LIN {X 72.334,Y 67.048,Z 77.329,A 180.000,B 0.000,C 180.000} C_DIS
LIN {X 72.380,Y 66.990,Z 77.327,A 180.000,B 0.000,C 180.000} C_DIS
LIN {X 72.424,Y 66.930,Z 77.324,A 180.000,B 0.000,C 180.000} C_DIS
LIN {X 72.502,Y 66.814,Z 77.319,A 180.000,B 0.000,C 180.000} C_DIS
LIN {X 72.574,Y 66.694,Z 77.315,A 180.000,B 0.000,C 180.000} C_DIS
LIN {X 72.610,Y 66.630,Z 77.312,A 180.000,B 0.000,C 180.000} C_DIS
LIN {X 72.644,Y 66.564,Z 77.309,A 180.000,B 0.000,C 180.000} C_DIS
LIN {X 72.676,Y 66.497,Z 77.307,A 180.000,B 0.000,C 180.000} C_DIS
LIN {X 72.706,Y 66.429,Z 77.304,A 180.000,B 0.000,C 180.000} C_DIS
LIN {X 72.757,Y 66.302,Z 77.299,A 180.000,B 0.000,C 180.000} C_DIS
LIN {X 72.800,Y 66.173,Z 77.295,A 180.000,B 0.000,C 180.000} C_DIS
LIN {X 72.838,Y 66.038,Z 77.290,A 180.000,B 0.000,C 180.000} C_DIS
LIN {X 72.869,Y 65.902,Z 77.285,A 180.000,B 0.000,C 180.000} C_DIS
LIN {X 72.882,Y 65.831,Z 77.282,A 180.000,B 0.000,C 180.000} C_DIS
LIN {X 72.893,Y 65.760,Z 77.280,A 180.000,B 0.000,C 180.000} C_DIS
LIN {X 72.901,Y 65.688,Z 77.277,A 180.000,B 0.000,C 180.000} C_DIS
LIN {X 72.908,Y 65.617,Z 77.275,A 180.000,B 0.000,C 180.000} C_DIS
LIN {X 72.916,Y 65.480,Z 77.270,A 180.000,B 0.000,C 180.000} C_DIS
LIN {X 72.916,Y 65.344,Z 77.265,A 180.000,B 0.000,C 180.000} C_DIS
LIN {X 72.909,Y 65.208,Z 77.261,A 180.000,B 0.000,C 180.000} C_DIS
LIN {X 72.895,Y 65.072,Z 77.256,A 180.000,B 0.000,C 180.000} C_DIS
LIN {X 72.873,Y 64.933,Z 77.251,A 180.000,B 0.000,C 180.000} C_DIS
LIN {X 72.842,Y 64.795,Z 77.246,A 180.000,B 0.000,C 180.000} C_DIS
LIN {X 72.823,Y 64.722,Z 77.243,A 180.000,B 0.000,C 180.000} C_DIS
LIN {X 72.802,Y 64.649,Z 77.241,A 180.000,B 0.000,C 180.000} C_DIS
LIN {X 72.759,Y 64.503,Z 77.235,A 180.000,B 0.000,C 180.000} C_DIS
LIN {X 72.737,Y 64.427,Z 77.233,A 180.000,B 0.000,C 180.000} C_DIS
LIN {X 72.715,Y 64.352,Z 77.230,A 180.000,B 0.000,C 180.000} C_DIS
LIN {X 72.693,Y 64.276,Z 77.227,A 180.000,B 0.000,C 180.000} C_DIS
LIN {X 72.670,Y 64.201,Z 77.224,A 180.000,B 0.000,C 180.000} C_DIS
LIN {X 72.648,Y 64.125,Z 77.222,A 180.000,B 0.000,C 180.000} C_DIS
LIN {X 72.626,Y 64.049,Z 77.219,A 180.000,B 0.000,C 180.000} C_DIS
LIN {X 72.604,Y 63.974,Z 77.216,A 180.000,B 0.000,C 180.000} C_DIS
LIN {X 72.582,Y 63.898,Z 77.213,A 180.000,B 0.000,C 180.000} C_DIS
LIN {X 72.560,Y 63.822,Z 77.211,A 180.000,B 0.000,C 180.000} C_DIS
LIN {X 72.537,Y 63.747,Z 77.208,A 180.000,B 0.000,C 180.000} C_DIS
LIN {X 72.515,Y 63.671,Z 77.205,A 180.000,B 0.000,C 180.000} C_DIS
LIN {X 72.493,Y 63.596,Z 77.202,A 180.000,B 0.000,C 180.000} C_DIS
LIN {X 72.471,Y 63.520,Z 77.200,A 180.000,B 0.000,C 180.000} C_DIS
LIN {X 72.449,Y 63.444,Z 77.197,A 180.000,B 0.000,C 180.000} C_DIS
LIN {X 72.427,Y 63.369,Z 77.194,A 180.000,B 0.000,C 180.000} C_DIS
LIN {X 72.404,Y 63.293,Z 77.191,A 180.000,B 0.000,C 180.000} C_DIS
LIN {X 72.382,Y 63.217,Z 77.189,A 180.000,B 0.000,C 180.000} C_DIS
LIN {X 72.360,Y 63.142,Z 77.186,A 180.000,B 0.000,C 180.000} C_DIS
LIN {X 72.338,Y 63.066,Z 77.183,A 180.000,B 0.000,C 180.000} C_DIS
LIN {X 72.316,Y 62.991,Z 77.180,A 180.000,B 0.000,C 180.000} C_DIS
LIN {X 72.293,Y 62.915,Z 77.178,A 180.000,B 0.000,C 180.000} C_DIS
LIN {X 72.271,Y 62.839,Z 77.175,A 180.000,B 0.000,C 180.000} C_DIS
LIN {X 72.249,Y 62.764,Z 77.172,A 180.000,B 0.000,C 180.000} C_DIS
LIN {X 72.227,Y 62.688,Z 77.170,A 180.000,B 0.000,C 180.000} C_DIS
LIN {X 72.204,Y 62.613,Z 77.167,A 180.000,B 0.000,C 180.000} C_DIS
LIN {X 72.182,Y 62.537,Z 77.165,A 180.000,B 0.000,C 180.000} C_DIS
LIN {X 72.160,Y 62.461,Z 77.162,A 180.000,B 0.000,C 180.000} C_DIS
LIN {X 72.137,Y 62.386,Z 77.159,A 180.000,B 0.000,C 180.000} C_DIS
LIN {X 72.115,Y 62.310,Z 77.157,A 180.000,B 0.000,C 180.000} C_DIS
LIN {X 72.093,Y 62.235,Z 77.154,A 180.000,B 0.000,C 180.000} C_DIS
LIN {X 72.070,Y 62.159,Z 77.152,A 180.000,B 0.000,C 180.000} C_DIS
LIN {X 72.048,Y 62.084,Z 77.149,A 180.000,B 0.000,C 180.000} C_DIS
LIN {X 72.003,Y 61.932,Z 77.144,A 180.000,B 0.000,C 180.000} C_DIS
LIN {X 71.958,Y 61.781,Z 77.139,A 180.000,B 0.000,C 180.000} C_DIS
LIN {X 71.913,Y 61.630,Z 77.134,A 180.000,B 0.000,C 180.000} C_DIS
LIN {X 71.868,Y 61.479,Z 77.130,A 180.000,B 0.000,C 180.000} C_DIS
LIN {X 71.823,Y 61.328,Z 77.125,A 180.000,B 0.000,C 180.000} C_DIS
LIN {X 71.777,Y 61.177,Z 77.120,A 180.000,B 0.000,C 180.000} C_DIS
LIN {X 71.732,Y 61.027,Z 77.116,A 180.000,B 0.000,C 180.000} C_DIS
LIN {X 71.687,Y 60.876,Z 77.111,A 180.000,B 0.000,C 180.000} C_DIS
LIN {X 71.641,Y 60.725,Z 77.107,A 180.000,B 0.000,C 180.000} C_DIS
LIN {X 71.596,Y 60.574,Z 77.102,A 180.000,B 0.000,C 180.000} C_DIS
LIN {X 71.550,Y 60.423,Z 77.098,A 180.000,B 0.000,C 180.000} C_DIS
LIN {X 71.504,Y 60.272,Z 77.094,A 180.000,B 0.000,C 180.000} C_DIS
LIN {X 71.458,Y 60.122,Z 77.090,A 180.000,B 0.000,C 180.000} C_DIS
LIN {X 71.412,Y 59.971,Z 77.086,A 180.000,B 0.000,C 180.000} C_DIS
LIN {X 71.366,Y 59.820,Z 77.082,A 180.000,B 0.000,C 180.000} C_DIS
LIN {X 71.320,Y 59.669,Z 77.078,A 180.000,B 0.000,C 180.000} C_DIS
LIN {X 71.274,Y 59.519,Z 77.074,A 180.000,B 0.000,C 180.000} C_DIS
LIN {X 71.228,Y 59.368,Z 77.070,A 180.000,B 0.000,C 180.000} C_DIS
LIN {X 71.182,Y 59.218,Z 77.066,A 180.000,B 0.000,C 180.000} C_DIS
LIN {X 71.135,Y 59.067,Z 77.063,A 180.000,B 0.000,C 180.000} C_DIS
LIN {X 71.089,Y 58.917,Z 77.059,A 180.000,B 0.000,C 180.000} C_DIS
LIN {X 71.042,Y 58.766,Z 77.056,A 180.000,B 0.000,C 180.000} C_DIS
LIN {X 70.995,Y 58.616,Z 77.053,A 180.000,B 0.000,C 180.000} C_DIS
LIN {X 70.948,Y 58.465,Z 77.049,A 180.000,B 0.000,C 180.000} C_DIS
LIN {X 70.901,Y 58.315,Z 77.046,A 180.000,B 0.000,C 180.000} C_DIS
LIN {X 70.854,Y 58.164,Z 77.043,A 180.000,B 0.000,C 180.000} C_DIS
LIN {X 70.807,Y 58.014,Z 77.040,A 180.000,B 0.000,C 180.000} C_DIS
LIN {X 70.760,Y 57.864,Z 77.037,A 180.000,B 0.000,C 180.000} C_DIS
LIN {X 70.713,Y 57.714,Z 77.035,A 180.000,B 0.000,C 180.000} C_DIS
LIN {X 70.665,Y 57.563,Z 77.032,A 180.000,B 0.000,C 180.000} C_DIS
LIN {X 70.618,Y 57.413,Z 77.029,A 180.000,B 0.000,C 180.000} C_DIS
LIN {X 70.570,Y 57.263,Z 77.027,A 180.000,B 0.000,C 180.000} C_DIS
LIN {X 70.474,Y 56.963,Z 77.022,A 180.000,B 0.000,C 180.000} C_DIS
LIN {X 70.378,Y 56.663,Z 77.018,A 180.000,B 0.000,C 180.000} C_DIS
LIN {X 70.282,Y 56.363,Z 77.014,A 180.000,B 0.000,C 180.000} C_DIS
LIN {X 70.185,Y 56.063,Z 77.011,A 180.000,B 0.000,C 180.000} C_DIS
LIN {X 70.087,Y 55.764,Z 77.008,A 180.000,B 0.000,C 180.000} C_DIS
LIN {X 69.989,Y 55.464,Z 77.006,A 180.000,B 0.000,C 180.000} C_DIS
LIN {X 69.891,Y 55.165,Z 77.004,A 180.000,B 0.000,C 180.000} C_DIS
LIN {X 69.792,Y 54.866,Z 77.002,A 180.000,B 0.000,C 180.000} C_DIS
LIN {X 69.693,Y 54.567,Z 77.001,A 180.000,B 0.000,C 180.000} C_DIS
LIN {X 69.593,Y 54.268,Z 77.000,A 180.000,B 0.000,C 180.000} C_DIS
LIN {X 69.512,Y 54.029,Z 77.000,A 180.000,B 0.000,C 180.000} C_DIS
; Cutting Move Starts
LIN {X 66.725,Y 45.768,Z 77.000,A 180.000,B 0.000,C 180.000} C_DIS
LIN {X 66.684,Y 45.647,Z 77.000,A 180.000,B 0.000,C 180.000} C_DIS
LIN {X 66.664,Y 45.590,Z 77.000,A 180.000,B 0.000,C 180.000} C_DIS
LIN {X 66.590,Y 45.411,Z 77.000,A 180.000,B 0.000,C 180.000} C_DIS
LIN {X 66.506,Y 45.243,Z 77.000,A 180.000,B 0.000,C 180.000} C_DIS
LIN {X 66.499,Y 45.232,Z 77.000,A 180.000,B 0.000,C 180.000} C_DIS
LIN {X 66.389,Y 45.053,Z 77.000,A 180.000,B 0.000,C 180.000} C_DIS
LIN {X 66.327,Y 44.965,Z 77.000,A 180.000,B 0.000,C 180.000} C_DIS
LIN {X 66.256,Y 44.874,Z 77.000,A 180.000,B 0.000,C 180.000} C_DIS
LIN {X 66.148,Y 44.750,Z 77.000,A 180.000,B 0.000,C 180.000} C_DIS
LIN {X 66.096,Y 44.696,Z 77.000,A 180.000,B 0.000,C 180.000} C_DIS
LIN {X 65.969,Y 44.576,Z 77.000,A 180.000,B 0.000,C 180.000} C_DIS
LIN {X 65.899,Y 44.517,Z 77.000,A 180.000,B 0.000,C 180.000} C_DIS
LIN {X 65.791,Y 44.433,Z 77.000,A 180.000,B 0.000,C 180.000} C_DIS
LIN {X 65.650,Y 44.338,Z 77.000,A 180.000,B 0.000,C 180.000} C_DIS
LIN {X 65.612,Y 44.314,Z 77.000,A 180.000,B 0.000,C 180.000} C_DIS
LIN {X 65.433,Y 44.216,Z 77.000,A 180.000,B 0.000,C 180.000} C_DIS
LIN {X 65.312,Y 44.159,Z 77.000,A 180.000,B 0.000,C 180.000} C_DIS
LIN {X 65.254,Y 44.135,Z 77.000,A 180.000,B 0.000,C 180.000} C_DIS
LIN {X 65.075,Y 44.071,Z 77.000,A 180.000,B 0.000,C 180.000} C_DIS
LIN {X 64.897,Y 44.021,Z 77.000,A 180.000,B 0.000,C 180.000} C_DIS
LIN {X 64.718,Y 43.986,Z 77.000,A 180.000,B 0.000,C 180.000} C_DIS
LIN {X 64.685,Y 43.981,Z 77.000,A 180.000,B 0.000,C 180.000} C_DIS
LIN {X 64.539,Y 43.963,Z 77.000,A 180.000,B 0.000,C 180.000} C_DIS
LIN {X 64.450,Y 43.957,Z 77.000,A 180.000,B 0.000,C 180.000} C_DIS
LIN {X 64.360,Y 43.954,Z 77.000,A 180.000,B 0.000,C 180.000} C_DIS
LIN {X 64.271,Y 43.954,Z 77.000,A 180.000,B 0.000,C 180.000} C_DIS
LIN {X 64.182,Y 43.957,Z 77.000,A 180.000,B 0.000,C 180.000} C_DIS
LIN {X 64.092,Y 43.964,Z 77.000,A 180.000,B 0.000,C 180.000} C_DIS
LIN {X 64.003,Y 43.973,Z 77.000,A 180.000,B 0.000,C 180.000} C_DIS
LIN {X 63.951,Y 43.981,Z 77.000,A 180.000,B 0.000,C 180.000} C_DIS
LIN {X 63.824,Y 44.003,Z 77.000,A 180.000,B 0.000,C 180.000} C_DIS
LIN {X 63.735,Y 44.022,Z 77.000,A 180.000,B 0.000,C 180.000} C_DIS
LIN {X 63.645,Y 44.046,Z 77.000,A 180.000,B 0.000,C 180.000} C_DIS
LIN {X 63.467,Y 44.102,Z 77.000,A 180.000,B 0.000,C 180.000} C_DIS
LIN {X 45.590,Y 50.133,Z 77.000,A 180.000,B 0.000,C 180.000} C_DIS
LIN {X 45.411,Y 50.194,Z 77.000,A 180.000,B 0.000,C 180.000} C_DIS
LIN {X 45.296,Y 50.238,Z 77.000,A 180.000,B 0.000,C 180.000} C_DIS
LIN {X 45.232,Y 50.265,Z 77.000,A 180.000,B 0.000,C 180.000} C_DIS
LIN {X 45.053,Y 50.353,Z 77.000,A 180.000,B 0.000,C 180.000} C_DIS
LIN {X 44.944,Y 50.416,Z 77.000,A 180.000,B 0.000,C 180.000} C_DIS
LIN {X 44.874,Y 50.461,Z 77.000,A 180.000,B 0.000,C 180.000} C_DIS
LIN {X 44.785,Y 50.522,Z 77.000,A 180.000,B 0.000,C 180.000} C_DIS
LIN {X 44.696,Y 50.590,Z 77.000,A 180.000,B 0.000,C 180.000} C_DIS
LIN {X 44.689,Y 50.595,Z 77.000,A 180.000,B 0.000,C 180.000} C_DIS
LIN {X 44.603,Y 50.667,Z 77.000,A 180.000,B 0.000,C 180.000} C_DIS
LIN {X 44.517,Y 50.746,Z 77.000,A 180.000,B 0.000,C 180.000} C_DIS
LIN {X 44.488,Y 50.774,Z 77.000,A 180.000,B 0.000,C 180.000} C_DIS
LIN {X 44.410,Y 50.855,Z 77.000,A 180.000,B 0.000,C 180.000} C_DIS
LIN {X 44.338,Y 50.936,Z 77.000,A 180.000,B 0.000,C 180.000} C_DIS
LIN {X 44.325,Y 50.953,Z 77.000,A 180.000,B 0.000,C 180.000} C_DIS
LIN {X 44.254,Y 51.042,Z 77.000,A 180.000,B 0.000,C 180.000} C_DIS
LIN {X 44.189,Y 51.131,Z 77.000,A 180.000,B 0.000,C 180.000} C_DIS
LIN {X 44.159,Y 51.176,Z 77.000,A 180.000,B 0.000,C 180.000} C_DIS
LIN {X 44.077,Y 51.310,Z 77.000,A 180.000,B 0.000,C 180.000} C_DIS
LIN {X 43.984,Y 51.489,Z 77.000,A 180.000,B 0.000,C 180.000} C_DIS
LIN {X 43.981,Y 51.497,Z 77.000,A 180.000,B 0.000,C 180.000} C_DIS
LIN {X 43.909,Y 51.668,Z 77.000,A 180.000,B 0.000,C 180.000} C_DIS
LIN {X 43.849,Y 51.847,Z 77.000,A 180.000,B 0.000,C 180.000} C_DIS
LIN {X 43.804,Y 52.025,Z 77.000,A 180.000,B 0.000,C 180.000} C_DIS
LIN {X 43.802,Y 52.035,Z 77.000,A 180.000,B 0.000,C 180.000} C_DIS
LIN {X 43.772,Y 52.204,Z 77.000,A 180.000,B 0.000,C 180.000} C_DIS
LIN {X 43.754,Y 52.383,Z 77.000,A 180.000,B 0.000,C 180.000} C_DIS
LIN {X 43.748,Y 52.562,Z 77.000,A 180.000,B 0.000,C 180.000} C_DIS
LIN {X 43.756,Y 52.740,Z 77.000,A 180.000,B 0.000,C 180.000} C_DIS
LIN {X 43.776,Y 52.919,Z 77.000,A 180.000,B 0.000,C 180.000} C_DIS
LIN {X 43.802,Y 53.064,Z 77.000,A 180.000,B 0.000,C 180.000} C_DIS
LIN {X 43.809,Y 53.098,Z 77.000,A 180.000,B 0.000,C 180.000} C_DIS
LIN {X 43.856,Y 53.277,Z 77.000,A 180.000,B 0.000,C 180.000} C_DIS
LIN {X 43.916,Y 53.455,Z 77.000,A 180.000,B 0.000,C 180.000} C_DIS
LIN {X 50.248,Y 72.226,Z 77.000,A 180.000,B 0.000,C 180.000} C_DIS
LIN {X 50.311,Y 72.405,Z 77.000,A 180.000,B 0.000,C 180.000} C_DIS
LIN {X 50.388,Y 72.584,Z 77.000,A 180.000,B 0.000,C 180.000} C_DIS
LIN {X 50.416,Y 72.640,Z 77.000,A 180.000,B 0.000,C 180.000} C_DIS
LIN {X 50.484,Y 72.763,Z 77.000,A 180.000,B 0.000,C 180.000} C_DIS
LIN {X 50.566,Y 72.891,Z 77.000,A 180.000,B 0.000,C 180.000} C_DIS
LIN {X 50.595,Y 72.936,Z 77.000,A 180.000,B 0.000,C 180.000} C_DIS
LIN {X 50.599,Y 72.941,Z 77.000,A 180.000,B 0.000,C 180.000} C_DIS
LIN {X 50.665,Y 73.031,Z 77.000,A 180.000,B 0.000,C 180.000} C_DIS
LIN {X 50.737,Y 73.120,Z 77.000,A 180.000,B 0.000,C 180.000} C_DIS
LIN {X 50.774,Y 73.162,Z 77.000,A 180.000,B 0.000,C 180.000} C_DIS
LIN {X 50.905,Y 73.299,Z 77.000,A 180.000,B 0.000,C 180.000} C_DIS
LIN {X 50.953,Y 73.343,Z 77.000,A 180.000,B 0.000,C 180.000} C_DIS
LIN {X 51.112,Y 73.478,Z 77.000,A 180.000,B 0.000,C 180.000} C_DIS
LIN {X 51.131,Y 73.493,Z 77.000,A 180.000,B 0.000,C 180.000} C_DIS
LIN {X 51.310,Y 73.616,Z 77.000,A 180.000,B 0.000,C 180.000} C_DIS
LIN {X 51.376,Y 73.656,Z 77.000,A 180.000,B 0.000,C 180.000} C_DIS
LIN {X 51.489,Y 73.719,Z 77.000,A 180.000,B 0.000,C 180.000} C_DIS
LIN {X 51.668,Y 73.803,Z 77.000,A 180.000,B 0.000,C 180.000} C_DIS
LIN {X 51.749,Y 73.835,Z 77.000,A 180.000,B 0.000,C 180.000} C_DIS
LIN {X 51.847,Y 73.870,Z 77.000,A 180.000,B 0.000,C 180.000} C_DIS
LIN {X 52.025,Y 73.923,Z 77.000,A 180.000,B 0.000,C 180.000} C_DIS
LIN {X 52.204,Y 73.961,Z 77.000,A 180.000,B 0.000,C 180.000} C_DIS
LIN {X 52.383,Y 73.987,Z 77.000,A 180.000,B 0.000,C 180.000} C_DIS
LIN {X 52.562,Y 73.999,Z 77.000,A 180.000,B 0.000,C 180.000} C_DIS
LIN {X 52.740,Y 73.998,Z 77.000,A 180.000,B 0.000,C 180.000} C_DIS
LIN {X 52.919,Y 73.985,Z 77.000,A 180.000,B 0.000,C 180.000} C_DIS
LIN {X 53.098,Y 73.958,Z 77.000,A 180.000,B 0.000,C 180.000} C_DIS
LIN {X 53.277,Y 73.918,Z 77.000,A 180.000,B 0.000,C 180.000} C_DIS
LIN {X 53.455,Y 73.864,Z 77.000,A 180.000,B 0.000,C 180.000} C_DIS
LIN {X 71.511,Y 67.773,Z 77.000,A 180.000,B 0.000,C 180.000} C_DIS
LIN {X 71.556,Y 67.757,Z 77.000,A 180.000,B 0.000,C 180.000} C_DIS
LIN {X 71.623,Y 67.732,Z 77.000,A 180.000,B 0.000,C 180.000} C_DIS
LIN {X 71.690,Y 67.705,Z 77.000,A 180.000,B 0.000,C 180.000} C_DIS
LIN {X 71.779,Y 67.664,Z 77.000,A 180.000,B 0.000,C 180.000} C_DIS
LIN {X 71.869,Y 67.620,Z 77.000,A 180.000,B 0.000,C 180.000} C_DIS
LIN {X 71.945,Y 67.578,Z 77.000,A 180.000,B 0.000,C 180.000} C_DIS
LIN {X 72.048,Y 67.517,Z 77.000,A 180.000,B 0.000,C 180.000} C_DIS
LIN {X 72.132,Y 67.461,Z 77.000,A 180.000,B 0.000,C 180.000} C_DIS
LIN {X 72.217,Y 67.399,Z 77.000,A 180.000,B 0.000,C 180.000} C_DIS
LIN {X 72.226,Y 67.393,Z 77.000,A 180.000,B 0.000,C 180.000} C_DIS
LIN {X 72.316,Y 67.321,Z 77.000,A 180.000,B 0.000,C 180.000} C_DIS
LIN {X 72.405,Y 67.243,Z 77.000,A 180.000,B 0.000,C 180.000} C_DIS
LIN {X 72.429,Y 67.221,Z 77.000,A 180.000,B 0.000,C 180.000} C_DIS
LIN {X 72.510,Y 67.140,Z 77.000,A 180.000,B 0.000,C 180.000} C_DIS
LIN {X 72.584,Y 67.060,Z 77.000,A 180.000,B 0.000,C 180.000} C_DIS
LIN {X 72.600,Y 67.042,Z 77.000,A 180.000,B 0.000,C 180.000} C_DIS
LIN {X 72.674,Y 66.953,Z 77.000,A 180.000,B 0.000,C 180.000} C_DIS
LIN {X 72.741,Y 66.863,Z 77.000,A 180.000,B 0.000,C 180.000} C_DIS
LIN {X 72.763,Y 66.833,Z 77.000,A 180.000,B 0.000,C 180.000} C_DIS
LIN {X 72.858,Y 66.684,Z 77.000,A 180.000,B 0.000,C 180.000} C_DIS
LIN {X 72.941,Y 66.534,Z 77.000,A 180.000,B 0.000,C 180.000} C_DIS
LIN {X 72.955,Y 66.506,Z 77.000,A 180.000,B 0.000,C 180.000} C_DIS
LIN {X 73.035,Y 66.327,Z 77.000,A 180.000,B 0.000,C 180.000} C_DIS
LIN {X 73.098,Y 66.148,Z 77.000,A 180.000,B 0.000,C 180.000} C_DIS
LIN {X 73.120,Y 66.072,Z 77.000,A 180.000,B 0.000,C 180.000} C_DIS
LIN {X 73.146,Y 65.969,Z 77.000,A 180.000,B 0.000,C 180.000} C_DIS
LIN {X 73.181,Y 65.791,Z 77.000,A 180.000,B 0.000,C 180.000} C_DIS
LIN {X 73.202,Y 65.612,Z 77.000,A 180.000,B 0.000,C 180.000} C_DIS
LIN {X 73.211,Y 65.433,Z 77.000,A 180.000,B 0.000,C 180.000} C_DIS
LIN {X 73.207,Y 65.254,Z 77.000,A 180.000,B 0.000,C 180.000} C_DIS
LIN {X 73.189,Y 65.075,Z 77.000,A 180.000,B 0.000,C 180.000} C_DIS
LIN {X 73.159,Y 64.897,Z 77.000,A 180.000,B 0.000,C 180.000} C_DIS
LIN {X 73.120,Y 64.736,Z 77.000,A 180.000,B 0.000,C 180.000} C_DIS
LIN {X 73.115,Y 64.718,Z 77.000,A 180.000,B 0.000,C 180.000} C_DIS
LIN {X 73.058,Y 64.539,Z 77.000,A 180.000,B 0.000,C 180.000} C_DIS
LIN {X 69.512,Y 54.029,Z 77.000,A 180.000,B 0.000,C 180.000} C_DIS
; Link Move Starts
LIN {X 69.412,Y 53.731,Z 77.000,A 180.000,B 0.000,C 180.000} C_DIS
LIN {X 69.312,Y 53.432,Z 76.999,A 180.000,B 0.000,C 180.000} C_DIS
LIN {X 69.212,Y 53.133,Z 76.998,A 180.000,B 0.000,C 180.000} C_DIS
LIN {X 69.114,Y 52.834,Z 76.996,A 180.000,B 0.000,C 180.000} C_DIS
LIN {X 69.015,Y 52.535,Z 76.994,A 180.000,B 0.000,C 180.000} C_DIS
LIN {X 68.917,Y 52.235,Z 76.991,A 180.000,B 0.000,C 180.000} C_DIS
LIN {X 68.820,Y 51.936,Z 76.988,A 180.000,B 0.000,C 180.000} C_DIS
LIN {X 68.723,Y 51.636,Z 76.985,A 180.000,B 0.000,C 180.000} C_DIS
LIN {X 68.627,Y 51.336,Z 76.981,A 180.000,B 0.000,C 180.000} C_DIS
LIN {X 68.531,Y 51.036,Z 76.977,A 180.000,B 0.000,C 180.000} C_DIS
LIN {X 68.435,Y 50.736,Z 76.972,A 180.000,B 0.000,C 180.000} C_DIS
LIN {X 68.388,Y 50.586,Z 76.969,A 180.000,B 0.000,C 180.000} C_DIS
LIN {X 68.340,Y 50.435,Z 76.967,A 180.000,B 0.000,C 180.000} C_DIS
LIN {X 68.293,Y 50.285,Z 76.964,A 180.000,B 0.000,C 180.000} C_DIS
LIN {X 68.245,Y 50.135,Z 76.961,A 180.000,B 0.000,C 180.000} C_DIS
LIN {X 68.198,Y 49.985,Z 76.959,A 180.000,B 0.000,C 180.000} C_DIS
LIN {X 68.151,Y 49.834,Z 76.956,A 180.000,B 0.000,C 180.000} C_DIS
LIN {X 68.104,Y 49.684,Z 76.952,A 180.000,B 0.000,C 180.000} C_DIS
LIN {X 68.057,Y 49.534,Z 76.949,A 180.000,B 0.000,C 180.000} C_DIS
LIN {X 68.010,Y 49.383,Z 76.946,A 180.000,B 0.000,C 180.000} C_DIS
LIN {X 67.964,Y 49.233,Z 76.943,A 180.000,B 0.000,C 180.000} C_DIS
LIN {X 67.917,Y 49.082,Z 76.939,A 180.000,B 0.000,C 180.000} C_DIS
LIN {X 67.871,Y 48.932,Z 76.936,A 180.000,B 0.000,C 180.000} C_DIS
LIN {X 67.824,Y 48.781,Z 76.932,A 180.000,B 0.000,C 180.000} C_DIS
LIN {X 67.778,Y 48.630,Z 76.928,A 180.000,B 0.000,C 180.000} C_DIS
LIN {X 67.732,Y 48.480,Z 76.925,A 180.000,B 0.000,C 180.000} C_DIS
LIN {X 67.686,Y 48.329,Z 76.921,A 180.000,B 0.000,C 180.000} C_DIS
LIN {X 67.639,Y 48.178,Z 76.917,A 180.000,B 0.000,C 180.000} C_DIS
LIN {X 67.594,Y 48.028,Z 76.913,A 180.000,B 0.000,C 180.000} C_DIS
LIN {X 67.548,Y 47.877,Z 76.909,A 180.000,B 0.000,C 180.000} C_DIS
LIN {X 67.502,Y 47.726,Z 76.905,A 180.000,B 0.000,C 180.000} C_DIS
LIN {X 67.456,Y 47.575,Z 76.900,A 180.000,B 0.000,C 180.000} C_DIS
LIN {X 67.411,Y 47.425,Z 76.896,A 180.000,B 0.000,C 180.000} C_DIS
LIN {X 67.365,Y 47.274,Z 76.892,A 180.000,B 0.000,C 180.000} C_DIS
LIN {X 67.320,Y 47.123,Z 76.887,A 180.000,B 0.000,C 180.000} C_DIS
LIN {X 67.274,Y 46.972,Z 76.883,A 180.000,B 0.000,C 180.000} C_DIS
LIN {X 67.229,Y 46.821,Z 76.878,A 180.000,B 0.000,C 180.000} C_DIS
LIN {X 67.184,Y 46.670,Z 76.873,A 180.000,B 0.000,C 180.000} C_DIS
LIN {X 67.139,Y 46.519,Z 76.869,A 180.000,B 0.000,C 180.000} C_DIS
LIN {X 67.093,Y 46.368,Z 76.864,A 180.000,B 0.000,C 180.000} C_DIS
LIN {X 67.048,Y 46.217,Z 76.859,A 180.000,B 0.000,C 180.000} C_DIS
LIN {X 67.004,Y 46.066,Z 76.854,A 180.000,B 0.000,C 180.000} C_DIS
LIN {X 66.981,Y 45.990,Z 76.851,A 180.000,B 0.000,C 180.000} C_DIS
LIN {X 66.959,Y 45.915,Z 76.849,A 180.000,B 0.000,C 180.000} C_DIS
LIN {X 66.936,Y 45.840,Z 76.846,A 180.000,B 0.000,C 180.000} C_DIS
LIN {X 66.914,Y 45.765,Z 76.844,A 180.000,B 0.000,C 180.000} C_DIS
LIN {X 66.892,Y 45.691,Z 76.841,A 180.000,B 0.000,C 180.000} C_DIS
LIN {X 66.870,Y 45.616,Z 76.839,A 180.000,B 0.000,C 180.000} C_DIS
LIN {X 66.843,Y 45.528,Z 76.836,A 180.000,B 0.000,C 180.000} C_DIS
LIN {X 66.813,Y 45.441,Z 76.832,A 180.000,B 0.000,C 180.000} C_DIS
LIN {X 66.771,Y 45.333,Z 76.828,A 180.000,B 0.000,C 180.000} C_DIS
LIN {X 66.724,Y 45.227,Z 76.824,A 180.000,B 0.000,C 180.000} C_DIS
LIN {X 66.687,Y 45.153,Z 76.821,A 180.000,B 0.000,C 180.000} C_DIS
LIN {X 66.647,Y 45.080,Z 76.818,A 180.000,B 0.000,C 180.000} C_DIS
LIN {X 66.588,Y 44.979,Z 76.814,A 180.000,B 0.000,C 180.000} C_DIS
LIN {X 66.523,Y 44.881,Z 76.810,A 180.000,B 0.000,C 180.000} C_DIS
LIN {X 66.459,Y 44.792,Z 76.806,A 180.000,B 0.000,C 180.000} C_DIS
LIN {X 66.391,Y 44.707,Z 76.803,A 180.000,B 0.000,C 180.000} C_DIS
LIN {X 66.320,Y 44.626,Z 76.799,A 180.000,B 0.000,C 180.000} C_DIS
LIN {X 66.246,Y 44.549,Z 76.795,A 180.000,B 0.000,C 180.000} C_DIS
LIN {X 66.164,Y 44.471,Z 76.791,A 180.000,B 0.000,C 180.000} C_DIS
LIN {X 66.079,Y 44.396,Z 76.787,A 180.000,B 0.000,C 180.000} C_DIS
LIN {X 65.972,Y 44.313,Z 76.783,A 180.000,B 0.000,C 180.000} C_DIS
LIN {X 65.861,Y 44.237,Z 76.778,A 180.000,B 0.000,C 180.000} C_DIS
LIN {X 65.754,Y 44.171,Z 76.773,A 180.000,B 0.000,C 180.000} C_DIS
LIN {X 65.643,Y 44.110,Z 76.769,A 180.000,B 0.000,C 180.000} C_DIS
LIN {X 65.521,Y 44.052,Z 76.764,A 180.000,B 0.000,C 180.000} C_DIS
LIN {X 65.396,Y 44.002,Z 76.760,A 180.000,B 0.000,C 180.000} C_DIS
LIN {X 65.328,Y 43.977,Z 76.757,A 180.000,B 0.000,C 180.000} C_DIS
LIN {X 65.259,Y 43.955,Z 76.755,A 180.000,B 0.000,C 180.000} C_DIS
LIN {X 65.189,Y 43.935,Z 76.752,A 180.000,B 0.000,C 180.000} C_DIS
LIN {X 65.119,Y 43.917,Z 76.749,A 180.000,B 0.000,C 180.000} C_DIS
LIN {X 65.046,Y 43.901,Z 76.747,A 180.000,B 0.000,C 180.000} C_DIS
LIN {X 64.972,Y 43.887,Z 76.744,A 180.000,B 0.000,C 180.000} C_DIS
LIN {X 64.897,Y 43.876,Z 76.742,A 180.000,B 0.000,C 180.000} C_DIS
LIN {X 64.823,Y 43.867,Z 76.739,A 180.000,B 0.000,C 180.000} C_DIS
LIN {X 64.742,Y 43.860,Z 76.736,A 180.000,B 0.000,C 180.000} C_DIS
LIN {X 64.662,Y 43.856,Z 76.733,A 180.000,B 0.000,C 180.000} C_DIS
LIN {X 64.581,Y 43.854,Z 76.731,A 180.000,B 0.000,C 180.000} C_DIS
LIN {X 64.500,Y 43.856,Z 76.728,A 180.000,B 0.000,C 180.000} C_DIS
LIN {X 64.420,Y 43.860,Z 76.725,A 180.000,B 0.000,C 180.000} C_DIS
LIN {X 64.339,Y 43.867,Z 76.722,A 180.000,B 0.000,C 180.000} C_DIS
LIN {X 64.259,Y 43.877,Z 76.719,A 180.000,B 0.000,C 180.000} C_DIS
LIN {X 64.179,Y 43.890,Z 76.716,A 180.000,B 0.000,C 180.000} C_DIS
LIN {X 64.102,Y 43.905,Z 76.714,A 180.000,B 0.000,C 180.000} C_DIS
LIN {X 64.025,Y 43.922,Z 76.711,A 180.000,B 0.000,C 180.000} C_DIS
LIN {X 63.948,Y 43.943,Z 76.708,A 180.000,B 0.000,C 180.000} C_DIS
LIN {X 63.873,Y 43.966,Z 76.705,A 180.000,B 0.000,C 180.000} C_DIS
LIN {X 63.798,Y 43.991,Z 76.703,A 180.000,B 0.000,C 180.000} C_DIS
LIN {X 63.649,Y 44.041,Z 76.697,A 180.000,B 0.000,C 180.000} C_DIS
LIN {X 63.574,Y 44.066,Z 76.694,A 180.000,B 0.000,C 180.000} C_DIS
LIN {X 63.425,Y 44.116,Z 76.689,A 180.000,B 0.000,C 180.000} C_DIS
LIN {X 62.977,Y 44.267,Z 76.672,A 180.000,B 0.000,C 180.000} C_DIS
LIN {X 62.828,Y 44.318,Z 76.667,A 180.000,B 0.000,C 180.000} C_DIS
LIN {X 62.306,Y 44.494,Z 76.648,A 180.000,B 0.000,C 180.000} C_DIS
LIN {X 61.858,Y 44.645,Z 76.631,A 180.000,B 0.000,C 180.000} C_DIS
LIN {X 61.709,Y 44.695,Z 76.626,A 180.000,B 0.000,C 180.000} C_DIS
LIN {X 61.261,Y 44.846,Z 76.609,A 180.000,B 0.000,C 180.000} C_DIS
LIN {X 61.112,Y 44.897,Z 76.604,A 180.000,B 0.000,C 180.000} C_DIS
LIN {X 60.365,Y 45.148,Z 76.576,A 180.000,B 0.000,C 180.000} C_DIS
LIN {X 59.992,Y 45.274,Z 76.562,A 180.000,B 0.000,C 180.000} C_DIS
LIN {X 59.470,Y 45.451,Z 76.543,A 180.000,B 0.000,C 180.000} C_DIS
LIN {X 58.873,Y 45.652,Z 76.521,A 180.000,B 0.000,C 180.000} C_DIS
LIN {X 57.679,Y 46.055,Z 76.477,A 180.000,B 0.000,C 180.000} C_DIS
LIN {X 56.411,Y 46.483,Z 76.430,A 180.000,B 0.000,C 180.000} C_DIS
LIN {X 55.963,Y 46.634,Z 76.414,A 180.000,B 0.000,C 180.000} C_DIS
LIN {X 55.142,Y 46.911,Z 76.384,A 180.000,B 0.000,C 180.000} C_DIS
LIN {X 54.695,Y 47.062,Z 76.367,A 180.000,B 0.000,C 180.000} C_DIS
LIN {X 54.545,Y 47.112,Z 76.362,A 180.000,B 0.000,C 180.000} C_DIS
LIN {X 54.098,Y 47.263,Z 76.345,A 180.000,B 0.000,C 180.000} C_DIS
LIN {X 53.948,Y 47.313,Z 76.340,A 180.000,B 0.000,C 180.000} C_DIS
LIN {X 53.501,Y 47.464,Z 76.323,A 180.000,B 0.000,C 180.000} C_DIS
LIN {X 53.426,Y 47.489,Z 76.320,A 180.000,B 0.000,C 180.000} C_DIS
LIN {X 53.277,Y 47.540,Z 76.315,A 180.000,B 0.000,C 180.000} C_DIS
LIN {X 52.829,Y 47.691,Z 76.298,A 180.000,B 0.000,C 180.000} C_DIS
LIN {X 52.680,Y 47.741,Z 76.293,A 180.000,B 0.000,C 180.000} C_DIS
LIN {X 52.232,Y 47.892,Z 76.276,A 180.000,B 0.000,C 180.000} C_DIS
LIN {X 52.083,Y 47.943,Z 76.271,A 180.000,B 0.000,C 180.000} C_DIS
LIN {X 51.859,Y 48.018,Z 76.263,A 180.000,B 0.000,C 180.000} C_DIS
LIN {X 51.710,Y 48.068,Z 76.257,A 180.000,B 0.000,C 180.000} C_DIS
LIN {X 51.635,Y 48.094,Z 76.254,A 180.000,B 0.000,C 180.000} C_DIS
LIN {X 51.486,Y 48.144,Z 76.249,A 180.000,B 0.000,C 180.000} C_DIS
LIN {X 51.262,Y 48.219,Z 76.241,A 180.000,B 0.000,C 180.000} C_DIS
LIN {X 51.113,Y 48.270,Z 76.235,A 180.000,B 0.000,C 180.000} C_DIS
LIN {X 51.038,Y 48.295,Z 76.232,A 180.000,B 0.000,C 180.000} C_DIS
LIN {X 50.889,Y 48.345,Z 76.227,A 180.000,B 0.000,C 180.000} C_DIS
LIN {X 50.665,Y 48.421,Z 76.219,A 180.000,B 0.000,C 180.000} C_DIS
LIN {X 50.516,Y 48.471,Z 76.213,A 180.000,B 0.000,C 180.000} C_DIS
LIN {X 50.441,Y 48.496,Z 76.210,A 180.000,B 0.000,C 180.000} C_DIS
LIN {X 50.292,Y 48.547,Z 76.205,A 180.000,B 0.000,C 180.000} C_DIS
LIN {X 50.068,Y 48.622,Z 76.197,A 180.000,B 0.000,C 180.000} C_DIS
LIN {X 49.919,Y 48.673,Z 76.191,A 180.000,B 0.000,C 180.000} C_DIS
LIN {X 49.770,Y 48.723,Z 76.186,A 180.000,B 0.000,C 180.000} C_DIS
LIN {X 49.620,Y 48.773,Z 76.180,A 180.000,B 0.000,C 180.000} C_DIS
LIN {X 49.471,Y 48.824,Z 76.175,A 180.000,B 0.000,C 180.000} C_DIS
LIN {X 49.322,Y 48.874,Z 76.170,A 180.000,B 0.000,C 180.000} C_DIS
LIN {X 49.173,Y 48.924,Z 76.164,A 180.000,B 0.000,C 180.000} C_DIS
LIN {X 49.098,Y 48.949,Z 76.162,A 180.000,B 0.000,C 180.000} C_DIS
LIN {X 49.024,Y 48.975,Z 76.159,A 180.000,B 0.000,C 180.000} C_DIS
LIN {X 48.949,Y 49.000,Z 76.157,A 180.000,B 0.000,C 180.000} C_DIS
LIN {X 48.874,Y 49.025,Z 76.154,A 180.000,B 0.000,C 180.000} C_DIS
LIN {X 48.800,Y 49.050,Z 76.152,A 180.000,B 0.000,C 180.000} C_DIS
LIN {X 48.725,Y 49.075,Z 76.149,A 180.000,B 0.000,C 180.000} C_DIS
LIN {X 48.650,Y 49.101,Z 76.147,A 180.000,B 0.000,C 180.000} C_DIS
LIN {X 48.501,Y 49.151,Z 76.142,A 180.000,B 0.000,C 180.000} C_DIS
LIN {X 48.352,Y 49.201,Z 76.137,A 180.000,B 0.000,C 180.000} C_DIS
LIN {X 48.203,Y 49.252,Z 76.132,A 180.000,B 0.000,C 180.000} C_DIS
LIN {X 48.053,Y 49.302,Z 76.127,A 180.000,B 0.000,C 180.000} C_DIS
LIN {X 47.904,Y 49.352,Z 76.122,A 180.000,B 0.000,C 180.000} C_DIS
LIN {X 47.755,Y 49.403,Z 76.118,A 180.000,B 0.000,C 180.000} C_DIS
LIN {X 47.606,Y 49.453,Z 76.113,A 180.000,B 0.000,C 180.000} C_DIS
LIN {X 47.457,Y 49.503,Z 76.109,A 180.000,B 0.000,C 180.000} C_DIS
LIN {X 47.307,Y 49.554,Z 76.104,A 180.000,B 0.000,C 180.000} C_DIS
LIN {X 47.158,Y 49.604,Z 76.100,A 180.000,B 0.000,C 180.000} C_DIS
LIN {X 47.009,Y 49.654,Z 76.096,A 180.000,B 0.000,C 180.000} C_DIS
LIN {X 46.860,Y 49.705,Z 76.092,A 180.000,B 0.000,C 180.000} C_DIS
LIN {X 46.710,Y 49.755,Z 76.087,A 180.000,B 0.000,C 180.000} C_DIS
LIN {X 46.561,Y 49.805,Z 76.083,A 180.000,B 0.000,C 180.000} C_DIS
LIN {X 46.412,Y 49.856,Z 76.080,A 180.000,B 0.000,C 180.000} C_DIS
LIN {X 46.263,Y 49.906,Z 76.076,A 180.000,B 0.000,C 180.000} C_DIS
LIN {X 46.113,Y 49.956,Z 76.072,A 180.000,B 0.000,C 180.000} C_DIS
LIN {X 45.964,Y 50.007,Z 76.068,A 180.000,B 0.000,C 180.000} C_DIS
LIN {X 45.815,Y 50.057,Z 76.065,A 180.000,B 0.000,C 180.000} C_DIS
LIN {X 45.666,Y 50.107,Z 76.061,A 180.000,B 0.000,C 180.000} C_DIS
LIN {X 45.516,Y 50.158,Z 76.058,A 180.000,B 0.000,C 180.000} C_DIS
LIN {X 45.368,Y 50.210,Z 76.054,A 180.000,B 0.000,C 180.000} C_DIS
LIN {X 45.222,Y 50.270,Z 76.051,A 180.000,B 0.000,C 180.000} C_DIS
LIN {X 45.081,Y 50.339,Z 76.048,A 180.000,B 0.000,C 180.000} C_DIS
LIN {X 44.944,Y 50.417,Z 76.045,A 180.000,B 0.000,C 180.000} C_DIS
LIN {X 44.812,Y 50.503,Z 76.042,A 180.000,B 0.000,C 180.000} C_DIS
LIN {X 44.686,Y 50.598,Z 76.039,A 180.000,B 0.000,C 180.000} C_DIS
LIN {X 44.566,Y 50.700,Z 76.036,A 180.000,B 0.000,C 180.000} C_DIS
LIN {X 44.453,Y 50.809,Z 76.033,A 180.000,B 0.000,C 180.000} C_DIS
LIN {X 44.347,Y 50.926,Z 76.031,A 180.000,B 0.000,C 180.000} C_DIS
LIN {X 44.249,Y 51.049,Z 76.028,A 180.000,B 0.000,C 180.000} C_DIS
LIN {X 44.158,Y 51.178,Z 76.026,A 180.000,B 0.000,C 180.000} C_DIS
LIN {X 44.076,Y 51.312,Z 76.023,A 180.000,B 0.000,C 180.000} C_DIS
LIN {X 44.002,Y 51.451,Z 76.021,A 180.000,B 0.000,C 180.000} C_DIS
LIN {X 43.938,Y 51.595,Z 76.019,A 180.000,B 0.000,C 180.000} C_DIS
LIN {X 43.882,Y 51.742,Z 76.017,A 180.000,B 0.000,C 180.000} C_DIS
LIN {X 43.836,Y 51.893,Z 76.015,A 180.000,B 0.000,C 180.000} C_DIS
LIN {X 43.799,Y 52.046,Z 76.013,A 180.000,B 0.000,C 180.000} C_DIS
LIN {X 43.773,Y 52.201,Z 76.012,A 180.000,B 0.000,C 180.000} C_DIS
LIN {X 43.756,Y 52.358,Z 76.010,A 180.000,B 0.000,C 180.000} C_DIS
LIN {X 43.749,Y 52.515,Z 76.009,A 180.000,B 0.000,C 180.000} C_DIS
LIN {X 43.751,Y 52.673,Z 76.007,A 180.000,B 0.000,C 180.000} C_DIS
LIN {X 43.764,Y 52.830,Z 76.006,A 180.000,B 0.000,C 180.000} C_DIS
LIN {X 43.787,Y 52.985,Z 76.005,A 180.000,B 0.000,C 180.000} C_DIS
LIN {X 43.819,Y 53.140,Z 76.004,A 180.000,B 0.000,C 180.000} C_DIS
LIN {X 43.861,Y 53.291,Z 76.003,A 180.000,B 0.000,C 180.000} C_DIS
LIN {X 43.961,Y 53.590,Z 76.002,A 180.000,B 0.000,C 180.000} C_DIS
LIN {X 44.062,Y 53.889,Z 76.001,A 180.000,B 0.000,C 180.000} C_DIS
LIN {X 44.162,Y 54.187,Z 76.000,A 180.000,B 0.000,C 180.000} C_DIS
LIN {X 44.217,Y 54.348,Z 76.000,A 180.000,B 0.000,C 180.000} C_DIS
; Cutting Move Starts
LIN {X 50.248,Y 72.226,Z 76.000,A 180.000,B 0.000,C 180.000} C_DIS
LIN {X 50.311,Y 72.405,Z 76.000,A 180.000,B 0.000,C 180.000} C_DIS
LIN {X 50.388,Y 72.584,Z 76.000,A 180.000,B 0.000,C 180.000} C_DIS
LIN {X 50.416,Y 72.640,Z 76.000,A 180.000,B 0.000,C 180.000} C_DIS
LIN {X 50.484,Y 72.763,Z 76.000,A 180.000,B 0.000,C 180.000} C_DIS
LIN {X 50.595,Y 72.936,Z 76.000,A 180.000,B 0.000,C 180.000} C_DIS
LIN {X 50.599,Y 72.941,Z 76.000,A 180.000,B 0.000,C 180.000} C_DIS
LIN {X 50.665,Y 73.031,Z 76.000,A 180.000,B 0.000,C 180.000} C_DIS
LIN {X 50.737,Y 73.120,Z 76.000,A 180.000,B 0.000,C 180.000} C_DIS
LIN {X 50.774,Y 73.162,Z 76.000,A 180.000,B 0.000,C 180.000} C_DIS
LIN {X 50.905,Y 73.299,Z 76.000,A 180.000,B 0.000,C 180.000} C_DIS
LIN {X 50.953,Y 73.343,Z 76.000,A 180.000,B 0.000,C 180.000} C_DIS
LIN {X 51.112,Y 73.478,Z 76.000,A 180.000,B 0.000,C 180.000} C_DIS
LIN {X 51.131,Y 73.493,Z 76.000,A 180.000,B 0.000,C 180.000} C_DIS
LIN {X 51.310,Y 73.616,Z 76.000,A 180.000,B 0.000,C 180.000} C_DIS
LIN {X 51.376,Y 73.656,Z 76.000,A 180.000,B 0.000,C 180.000} C_DIS
LIN {X 51.489,Y 73.719,Z 76.000,A 180.000,B 0.000,C 180.000} C_DIS
LIN {X 51.668,Y 73.803,Z 76.000,A 180.000,B 0.000,C 180.000} C_DIS
LIN {X 51.749,Y 73.835,Z 76.000,A 180.000,B 0.000,C 180.000} C_DIS
LIN {X 51.847,Y 73.870,Z 76.000,A 180.000,B 0.000,C 180.000} C_DIS
LIN {X 52.025,Y 73.923,Z 76.000,A 180.000,B 0.000,C 180.000} C_DIS
LIN {X 52.204,Y 73.961,Z 76.000,A 180.000,B 0.000,C 180.000} C_DIS
LIN {X 52.383,Y 73.987,Z 76.000,A 180.000,B 0.000,C 180.000} C_DIS
LIN {X 52.562,Y 73.999,Z 76.000,A 180.000,B 0.000,C 180.000} C_DIS
LIN {X 52.740,Y 73.998,Z 76.000,A 180.000,B 0.000,C 180.000} C_DIS
LIN {X 52.919,Y 73.985,Z 76.000,A 180.000,B 0.000,C 180.000} C_DIS
LIN {X 53.098,Y 73.958,Z 76.000,A 180.000,B 0.000,C 180.000} C_DIS
LIN {X 53.277,Y 73.918,Z 76.000,A 180.000,B 0.000,C 180.000} C_DIS
LIN {X 53.455,Y 73.864,Z 76.000,A 180.000,B 0.000,C 180.000} C_DIS
LIN {X 72.584,Y 67.411,Z 76.000,A 180.000,B 0.000,C 180.000} C_DIS
LIN {X 72.617,Y 67.399,Z 76.000,A 180.000,B 0.000,C 180.000} C_DIS
LIN {X 72.690,Y 67.373,Z 76.000,A 180.000,B 0.000,C 180.000} C_DIS
LIN {X 72.763,Y 67.344,Z 76.000,A 180.000,B 0.000,C 180.000} C_DIS
LIN {X 72.852,Y 67.305,Z 76.000,A 180.000,B 0.000,C 180.000} C_DIS
LIN {X 72.941,Y 67.262,Z 76.000,A 180.000,B 0.000,C 180.000} C_DIS
LIN {X 73.018,Y 67.221,Z 76.000,A 180.000,B 0.000,C 180.000} C_DIS
LIN {X 73.120,Y 67.161,Z 76.000,A 180.000,B 0.000,C 180.000} C_DIS
LIN {X 73.208,Y 67.104,Z 76.000,A 180.000,B 0.000,C 180.000} C_DIS
LIN {X 73.295,Y 67.042,Z 76.000,A 180.000,B 0.000,C 180.000} C_DIS
LIN {X 73.299,Y 67.039,Z 76.000,A 180.000,B 0.000,C 180.000} C_DIS
LIN {X 73.388,Y 66.969,Z 76.000,A 180.000,B 0.000,C 180.000} C_DIS
LIN {X 73.478,Y 66.892,Z 76.000,A 180.000,B 0.000,C 180.000} C_DIS
LIN {X 73.509,Y 66.863,Z 76.000,A 180.000,B 0.000,C 180.000} C_DIS
LIN {X 73.586,Y 66.789,Z 76.000,A 180.000,B 0.000,C 180.000} C_DIS
LIN {X 73.656,Y 66.714,Z 76.000,A 180.000,B 0.000,C 180.000} C_DIS
LIN {X 73.683,Y 66.684,Z 76.000,A 180.000,B 0.000,C 180.000} C_DIS
LIN {X 73.758,Y 66.595,Z 76.000,A 180.000,B 0.000,C 180.000} C_DIS
LIN {X 73.826,Y 66.506,Z 76.000,A 180.000,B 0.000,C 180.000} C_DIS
LIN {X 73.835,Y 66.493,Z 76.000,A 180.000,B 0.000,C 180.000} C_DIS
LIN {X 73.944,Y 66.327,Z 76.000,A 180.000,B 0.000,C 180.000} C_DIS
LIN {X 74.014,Y 66.204,Z 76.000,A 180.000,B 0.000,C 180.000} C_DIS
LIN {X 74.042,Y 66.148,Z 76.000,A 180.000,B 0.000,C 180.000} C_DIS
LIN {X 74.123,Y 65.969,Z 76.000,A 180.000,B 0.000,C 180.000} C_DIS
LIN {X 74.187,Y 65.791,Z 76.000,A 180.000,B 0.000,C 180.000} C_DIS
LIN {X 74.193,Y 65.772,Z 76.000,A 180.000,B 0.000,C 180.000} C_DIS
LIN {X 74.236,Y 65.612,Z 76.000,A 180.000,B 0.000,C 180.000} C_DIS
LIN {X 74.272,Y 65.433,Z 76.000,A 180.000,B 0.000,C 180.000} C_DIS
LIN {X 74.294,Y 65.254,Z 76.000,A 180.000,B 0.000,C 180.000} C_DIS
LIN {X 74.303,Y 65.075,Z 76.000,A 180.000,B 0.000,C 180.000} C_DIS
LIN {X 74.300,Y 64.897,Z 76.000,A 180.000,B 0.000,C 180.000} C_DIS
LIN {X 74.283,Y 64.718,Z 76.000,A 180.000,B 0.000,C 180.000} C_DIS
LIN {X 74.254,Y 64.539,Z 76.000,A 180.000,B 0.000,C 180.000} C_DIS
LIN {X 74.211,Y 64.360,Z 76.000,A 180.000,B 0.000,C 180.000} C_DIS
LIN {X 74.193,Y 64.299,Z 76.000,A 180.000,B 0.000,C 180.000} C_DIS
LIN {X 74.154,Y 64.182,Z 76.000,A 180.000,B 0.000,C 180.000} C_DIS
LIN {X 70.605,Y 53.661,Z 76.000,A 180.000,B 0.000,C 180.000} C_DIS
LIN {X 67.822,Y 45.411,Z 76.000,A 180.000,B 0.000,C 180.000} C_DIS
LIN {X 67.761,Y 45.232,Z 76.000,A 180.000,B 0.000,C 180.000} C_DIS
LIN {X 67.757,Y 45.222,Z 76.000,A 180.000,B 0.000,C 180.000} C_DIS
LIN {X 67.688,Y 45.053,Z 76.000,A 180.000,B 0.000,C 180.000} C_DIS
LIN {X 67.598,Y 44.874,Z 76.000,A 180.000,B 0.000,C 180.000} C_DIS
LIN {X 67.578,Y 44.839,Z 76.000,A 180.000,B 0.000,C 180.000} C_DIS
LIN {X 67.489,Y 44.696,Z 76.000,A 180.000,B 0.000,C 180.000} C_DIS
LIN {X 67.399,Y 44.570,Z 76.000,A 180.000,B 0.000,C 180.000} C_DIS
LIN {X 67.358,Y 44.517,Z 76.000,A 180.000,B 0.000,C 180.000} C_DIS
LIN {X 67.221,Y 44.360,Z 76.000,A 180.000,B 0.000,C 180.000} C_DIS
LIN {X 67.199,Y 44.338,Z 76.000,A 180.000,B 0.000,C 180.000} C_DIS
LIN {X 67.042,Y 44.190,Z 76.000,A 180.000,B 0.000,C 180.000} C_DIS
LIN {X 67.005,Y 44.159,Z 76.000,A 180.000,B 0.000,C 180.000} C_DIS
LIN {X 66.863,Y 44.050,Z 76.000,A 180.000,B 0.000,C 180.000} C_DIS
LIN {X 66.760,Y 43.981,Z 76.000,A 180.000,B 0.000,C 180.000} C_DIS
LIN {X 66.684,Y 43.934,Z 76.000,A 180.000,B 0.000,C 180.000} C_DIS
LIN {X 66.506,Y 43.837,Z 76.000,A 180.000,B 0.000,C 180.000} C_DIS
LIN {X 66.429,Y 43.802,Z 76.000,A 180.000,B 0.000,C 180.000} C_DIS
LIN {X 66.327,Y 43.759,Z 76.000,A 180.000,B 0.000,C 180.000} C_DIS
LIN {X 66.148,Y 43.696,Z 76.000,A 180.000,B 0.000,C 180.000} C_DIS
LIN {X 65.969,Y 43.648,Z 76.000,A 180.000,B 0.000,C 180.000} C_DIS
LIN {X 65.846,Y 43.623,Z 76.000,A 180.000,B 0.000,C 180.000} C_DIS
LIN {X 65.791,Y 43.614,Z 76.000,A 180.000,B 0.000,C 180.000} C_DIS
LIN {X 65.701,Y 43.602,Z 76.000,A 180.000,B 0.000,C 180.000} C_DIS
LIN {X 65.612,Y 43.593,Z 76.000,A 180.000,B 0.000,C 180.000} C_DIS
LIN {X 65.522,Y 43.587,Z 76.000,A 180.000,B 0.000,C 180.000} C_DIS
LIN {X 65.433,Y 43.585,Z 76.000,A 180.000,B 0.000,C 180.000} C_DIS
LIN {X 65.344,Y 43.586,Z 76.000,A 180.000,B 0.000,C 180.000} C_DIS
LIN {X 65.254,Y 43.590,Z 76.000,A 180.000,B 0.000,C 180.000} C_DIS
LIN {X 65.165,Y 43.597,Z 76.000,A 180.000,B 0.000,C 180.000} C_DIS
LIN {X 65.075,Y 43.607,Z 76.000,A 180.000,B 0.000,C 180.000} C_DIS
LIN {X 64.975,Y 43.623,Z 76.000,A 180.000,B 0.000,C 180.000} C_DIS
LIN {X 64.897,Y 43.638,Z 76.000,A 180.000,B 0.000,C 180.000} C_DIS
LIN {X 64.807,Y 43.659,Z 76.000,A 180.000,B 0.000,C 180.000} C_DIS
LIN {X 64.718,Y 43.683,Z 76.000,A 180.000,B 0.000,C 180.000} C_DIS
LIN {X 64.539,Y 43.740,Z 76.000,A 180.000,B 0.000,C 180.000} C_DIS
LIN {X 45.590,Y 50.133,Z 76.000,A 180.000,B 0.000,C 180.000} C_DIS
LIN {X 45.411,Y 50.194,Z 76.000,A 180.000,B 0.000,C 180.000} C_DIS
LIN {X 45.296,Y 50.238,Z 76.000,A 180.000,B 0.000,C 180.000} C_DIS
LIN {X 45.232,Y 50.265,Z 76.000,A 180.000,B 0.000,C 180.000} C_DIS
LIN {X 45.053,Y 50.353,Z 76.000,A 180.000,B 0.000,C 180.000} C_DIS
LIN {X 44.944,Y 50.416,Z 76.000,A 180.000,B 0.000,C 180.000} C_DIS
LIN {X 44.874,Y 50.461,Z 76.000,A 180.000,B 0.000,C 180.000} C_DIS
LIN {X 44.785,Y 50.522,Z 76.000,A 180.000,B 0.000,C 180.000} C_DIS
LIN {X 44.696,Y 50.590,Z 76.000,A 180.000,B 0.000,C 180.000} C_DIS
LIN {X 44.689,Y 50.595,Z 76.000,A 180.000,B 0.000,C 180.000} C_DIS
LIN {X 44.603,Y 50.667,Z 76.000,A 180.000,B 0.000,C 180.000} C_DIS
LIN {X 44.517,Y 50.746,Z 76.000,A 180.000,B 0.000,C 180.000} C_DIS
LIN {X 44.488,Y 50.774,Z 76.000,A 180.000,B 0.000,C 180.000} C_DIS
LIN {X 44.410,Y 50.855,Z 76.000,A 180.000,B 0.000,C 180.000} C_DIS
LIN {X 44.338,Y 50.936,Z 76.000,A 180.000,B 0.000,C 180.000} C_DIS
LIN {X 44.325,Y 50.953,Z 76.000,A 180.000,B 0.000,C 180.000} C_DIS
LIN {X 44.254,Y 51.042,Z 76.000,A 180.000,B 0.000,C 180.000} C_DIS
LIN {X 44.189,Y 51.131,Z 76.000,A 180.000,B 0.000,C 180.000} C_DIS
LIN {X 44.159,Y 51.176,Z 76.000,A 180.000,B 0.000,C 180.000} C_DIS
LIN {X 44.077,Y 51.310,Z 76.000,A 180.000,B 0.000,C 180.000} C_DIS
LIN {X 43.984,Y 51.489,Z 76.000,A 180.000,B 0.000,C 180.000} C_DIS
LIN {X 43.981,Y 51.497,Z 76.000,A 180.000,B 0.000,C 180.000} C_DIS
LIN {X 43.909,Y 51.668,Z 76.000,A 180.000,B 0.000,C 180.000} C_DIS
LIN {X 43.849,Y 51.847,Z 76.000,A 180.000,B 0.000,C 180.000} C_DIS
LIN {X 43.804,Y 52.025,Z 76.000,A 180.000,B 0.000,C 180.000} C_DIS
LIN {X 43.802,Y 52.035,Z 76.000,A 180.000,B 0.000,C 180.000} C_DIS
LIN {X 43.772,Y 52.204,Z 76.000,A 180.000,B 0.000,C 180.000} C_DIS
LIN {X 43.754,Y 52.383,Z 76.000,A 180.000,B 0.000,C 180.000} C_DIS
LIN {X 43.748,Y 52.562,Z 76.000,A 180.000,B 0.000,C 180.000} C_DIS
LIN {X 43.756,Y 52.740,Z 76.000,A 180.000,B 0.000,C 180.000} C_DIS
LIN {X 43.776,Y 52.919,Z 76.000,A 180.000,B 0.000,C 180.000} C_DIS
LIN {X 43.802,Y 53.064,Z 76.000,A 180.000,B 0.000,C 180.000} C_DIS
LIN {X 43.809,Y 53.098,Z 76.000,A 180.000,B 0.000,C 180.000} C_DIS
LIN {X 43.856,Y 53.277,Z 76.000,A 180.000,B 0.000,C 180.000} C_DIS
LIN {X 43.916,Y 53.455,Z 76.000,A 180.000,B 0.000,C 180.000} C_DIS
LIN {X 44.217,Y 54.348,Z 76.000,A 180.000,B 0.000,C 180.000} C_DIS
; Link Move Starts
LIN {X 44.317,Y 54.647,Z 76.000,A 180.000,B 0.000,C 180.000} C_DIS
LIN {X 44.418,Y 54.945,Z 75.999,A 180.000,B 0.000,C 180.000} C_DIS
LIN {X 44.519,Y 55.244,Z 75.998,A 180.000,B 0.000,C 180.000} C_DIS
LIN {X 44.619,Y 55.542,Z 75.996,A 180.000,B 0.000,C 180.000} C_DIS
LIN {X 44.720,Y 55.840,Z 75.994,A 180.000,B 0.000,C 180.000} C_DIS
LIN {X 44.821,Y 56.139,Z 75.991,A 180.000,B 0.000,C 180.000} C_DIS
LIN {X 44.922,Y 56.437,Z 75.988,A 180.000,B 0.000,C 180.000} C_DIS
LIN {X 45.022,Y 56.736,Z 75.985,A 180.000,B 0.000,C 180.000} C_DIS
LIN {X 45.123,Y 57.034,Z 75.981,A 180.000,B 0.000,C 180.000} C_DIS
LIN {X 45.224,Y 57.333,Z 75.977,A 180.000,B 0.000,C 180.000} C_DIS
LIN {X 45.324,Y 57.631,Z 75.972,A 180.000,B 0.000,C 180.000} C_DIS
LIN {X 45.375,Y 57.781,Z 75.969,A 180.000,B 0.000,C 180.000} C_DIS
LIN {X 45.425,Y 57.930,Z 75.967,A 180.000,B 0.000,C 180.000} C_DIS
LIN {X 45.475,Y 58.079,Z 75.964,A 180.000,B 0.000,C 180.000} C_DIS
LIN {X 45.526,Y 58.228,Z 75.961,A 180.000,B 0.000,C 180.000} C_DIS
LIN {X 45.576,Y 58.378,Z 75.959,A 180.000,B 0.000,C 180.000} C_DIS
LIN {X 45.626,Y 58.527,Z 75.956,A 180.000,B 0.000,C 180.000} C_DIS
LIN {X 45.677,Y 58.676,Z 75.952,A 180.000,B 0.000,C 180.000} C_DIS
LIN {X 45.727,Y 58.825,Z 75.949,A 180.000,B 0.000,C 180.000} C_DIS
LIN {X 45.777,Y 58.974,Z 75.946,A 180.000,B 0.000,C 180.000} C_DIS
LIN {X 45.828,Y 59.124,Z 75.943,A 180.000,B 0.000,C 180.000} C_DIS
LIN {X 45.878,Y 59.273,Z 75.939,A 180.000,B 0.000,C 180.000} C_DIS
LIN {X 45.928,Y 59.422,Z 75.936,A 180.000,B 0.000,C 180.000} C_DIS
LIN {X 45.979,Y 59.571,Z 75.932,A 180.000,B 0.000,C 180.000} C_DIS
LIN {X 46.029,Y 59.721,Z 75.928,A 180.000,B 0.000,C 180.000} C_DIS
LIN {X 46.079,Y 59.870,Z 75.925,A 180.000,B 0.000,C 180.000} C_DIS
LIN {X 46.130,Y 60.019,Z 75.921,A 180.000,B 0.000,C 180.000} C_DIS
LIN {X 46.180,Y 60.168,Z 75.917,A 180.000,B 0.000,C 180.000} C_DIS
LIN {X 46.231,Y 60.318,Z 75.913,A 180.000,B 0.000,C 180.000} C_DIS
LIN {X 46.281,Y 60.467,Z 75.909,A 180.000,B 0.000,C 180.000} C_DIS
LIN {X 46.331,Y 60.616,Z 75.905,A 180.000,B 0.000,C 180.000} C_DIS
LIN {X 46.382,Y 60.765,Z 75.900,A 180.000,B 0.000,C 180.000} C_DIS
LIN {X 46.432,Y 60.915,Z 75.896,A 180.000,B 0.000,C 180.000} C_DIS
LIN {X 46.482,Y 61.064,Z 75.892,A 180.000,B 0.000,C 180.000} C_DIS
LIN {X 46.533,Y 61.213,Z 75.887,A 180.000,B 0.000,C 180.000} C_DIS
LIN {X 46.583,Y 61.362,Z 75.883,A 180.000,B 0.000,C 180.000} C_DIS
LIN {X 46.633,Y 61.511,Z 75.878,A 180.000,B 0.000,C 180.000} C_DIS
LIN {X 46.684,Y 61.661,Z 75.873,A 180.000,B 0.000,C 180.000} C_DIS
LIN {X 46.734,Y 61.810,Z 75.869,A 180.000,B 0.000,C 180.000} C_DIS
LIN {X 46.784,Y 61.959,Z 75.864,A 180.000,B 0.000,C 180.000} C_DIS
LIN {X 46.835,Y 62.108,Z 75.859,A 180.000,B 0.000,C 180.000} C_DIS
LIN {X 46.885,Y 62.258,Z 75.854,A 180.000,B 0.000,C 180.000} C_DIS
LIN {X 46.910,Y 62.332,Z 75.851,A 180.000,B 0.000,C 180.000} C_DIS
LIN {X 46.935,Y 62.407,Z 75.849,A 180.000,B 0.000,C 180.000} C_DIS
LIN {X 46.961,Y 62.482,Z 75.846,A 180.000,B 0.000,C 180.000} C_DIS
LIN {X 46.986,Y 62.556,Z 75.844,A 180.000,B 0.000,C 180.000} C_DIS
LIN {X 47.011,Y 62.631,Z 75.841,A 180.000,B 0.000,C 180.000} C_DIS
LIN {X 47.036,Y 62.705,Z 75.839,A 180.000,B 0.000,C 180.000} C_DIS
LIN {X 47.061,Y 62.780,Z 75.836,A 180.000,B 0.000,C 180.000} C_DIS
LIN {X 47.112,Y 62.929,Z 75.831,A 180.000,B 0.000,C 180.000} C_DIS
LIN {X 47.162,Y 63.078,Z 75.825,A 180.000,B 0.000,C 180.000} C_DIS
LIN {X 47.212,Y 63.228,Z 75.820,A 180.000,B 0.000,C 180.000} C_DIS
LIN {X 47.263,Y 63.377,Z 75.815,A 180.000,B 0.000,C 180.000} C_DIS
LIN {X 47.313,Y 63.526,Z 75.809,A 180.000,B 0.000,C 180.000} C_DIS
LIN {X 47.338,Y 63.601,Z 75.807,A 180.000,B 0.000,C 180.000} C_DIS
LIN {X 47.388,Y 63.750,Z 75.801,A 180.000,B 0.000,C 180.000} C_DIS
LIN {X 47.464,Y 63.974,Z 75.793,A 180.000,B 0.000,C 180.000} C_DIS
LIN {X 47.514,Y 64.123,Z 75.787,A 180.000,B 0.000,C 180.000} C_DIS
LIN {X 47.539,Y 64.198,Z 75.785,A 180.000,B 0.000,C 180.000} C_DIS
LIN {X 47.590,Y 64.347,Z 75.779,A 180.000,B 0.000,C 180.000} C_DIS
LIN {X 47.665,Y 64.571,Z 75.771,A 180.000,B 0.000,C 180.000} C_DIS
LIN {X 47.716,Y 64.720,Z 75.765,A 180.000,B 0.000,C 180.000} C_DIS
LIN {X 47.741,Y 64.795,Z 75.763,A 180.000,B 0.000,C 180.000} C_DIS
LIN {X 47.791,Y 64.944,Z 75.757,A 180.000,B 0.000,C 180.000} C_DIS
LIN {X 47.867,Y 65.168,Z 75.749,A 180.000,B 0.000,C 180.000} C_DIS
LIN {X 47.917,Y 65.317,Z 75.743,A 180.000,B 0.000,C 180.000} C_DIS
LIN {X 47.942,Y 65.392,Z 75.741,A 180.000,B 0.000,C 180.000} C_DIS
LIN {X 47.993,Y 65.541,Z 75.735,A 180.000,B 0.000,C 180.000} C_DIS
LIN {X 48.068,Y 65.765,Z 75.727,A 180.000,B 0.000,C 180.000} C_DIS
LIN {X 48.118,Y 65.914,Z 75.721,A 180.000,B 0.000,C 180.000} C_DIS
LIN {X 48.144,Y 65.989,Z 75.719,A 180.000,B 0.000,C 180.000} C_DIS
LIN {X 48.194,Y 66.138,Z 75.713,A 180.000,B 0.000,C 180.000} C_DIS
LIN {X 48.345,Y 66.586,Z 75.697,A 180.000,B 0.000,C 180.000} C_DIS
LIN {X 48.395,Y 66.735,Z 75.691,A 180.000,B 0.000,C 180.000} C_DIS
LIN {X 48.546,Y 67.182,Z 75.675,A 180.000,B 0.000,C 180.000} C_DIS
LIN {X 48.597,Y 67.332,Z 75.669,A 180.000,B 0.000,C 180.000} C_DIS
LIN {X 48.773,Y 67.854,Z 75.650,A 180.000,B 0.000,C 180.000} C_DIS
LIN {X 48.924,Y 68.302,Z 75.633,A 180.000,B 0.000,C 180.000} C_DIS
LIN {X 48.974,Y 68.451,Z 75.628,A 180.000,B 0.000,C 180.000} C_DIS
LIN {X 49.125,Y 68.899,Z 75.611,A 180.000,B 0.000,C 180.000} C_DIS
LIN {X 49.176,Y 69.048,Z 75.606,A 180.000,B 0.000,C 180.000} C_DIS
LIN {X 49.427,Y 69.794,Z 75.578,A 180.000,B 0.000,C 180.000} C_DIS
LIN {X 49.553,Y 70.167,Z 75.565,A 180.000,B 0.000,C 180.000} C_DIS
LIN {X 49.704,Y 70.615,Z 75.548,A 180.000,B 0.000,C 180.000} C_DIS
LIN {X 50.258,Y 72.256,Z 75.488,A 180.000,B 0.000,C 180.000} C_DIS
LIN {X 50.283,Y 72.331,Z 75.485,A 180.000,B 0.000,C 180.000} C_DIS
LIN {X 50.311,Y 72.405,Z 75.482,A 180.000,B 0.000,C 180.000} C_DIS
LIN {X 50.340,Y 72.478,Z 75.479,A 180.000,B 0.000,C 180.000} C_DIS
LIN {X 50.372,Y 72.550,Z 75.477,A 180.000,B 0.000,C 180.000} C_DIS
LIN {X 50.407,Y 72.621,Z 75.474,A 180.000,B 0.000,C 180.000} C_DIS
LIN {X 50.443,Y 72.691,Z 75.471,A 180.000,B 0.000,C 180.000} C_DIS
LIN {X 50.482,Y 72.759,Z 75.468,A 180.000,B 0.000,C 180.000} C_DIS
LIN {X 50.522,Y 72.827,Z 75.466,A 180.000,B 0.000,C 180.000} C_DIS
LIN {X 50.565,Y 72.893,Z 75.463,A 180.000,B 0.000,C 180.000} C_DIS
LIN {X 50.610,Y 72.957,Z 75.460,A 180.000,B 0.000,C 180.000} C_DIS
LIN {X 50.657,Y 73.021,Z 75.457,A 180.000,B 0.000,C 180.000} C_DIS
LIN {X 50.706,Y 73.083,Z 75.455,A 180.000,B 0.000,C 180.000} C_DIS
LIN {X 50.757,Y 73.143,Z 75.452,A 180.000,B 0.000,C 180.000} C_DIS
LIN {X 50.809,Y 73.201,Z 75.449,A 180.000,B 0.000,C 180.000} C_DIS
LIN {X 50.864,Y 73.258,Z 75.446,A 180.000,B 0.000,C 180.000} C_DIS
LIN {X 50.920,Y 73.313,Z 75.444,A 180.000,B 0.000,C 180.000} C_DIS
LIN {X 50.978,Y 73.367,Z 75.441,A 180.000,B 0.000,C 180.000} C_DIS
LIN {X 51.038,Y 73.418,Z 75.438,A 180.000,B 0.000,C 180.000} C_DIS
LIN {X 51.099,Y 73.468,Z 75.435,A 180.000,B 0.000,C 180.000} C_DIS
LIN {X 51.162,Y 73.515,Z 75.433,A 180.000,B 0.000,C 180.000} C_DIS
LIN {X 51.226,Y 73.561,Z 75.430,A 180.000,B 0.000,C 180.000} C_DIS
LIN {X 51.292,Y 73.604,Z 75.427,A 180.000,B 0.000,C 180.000} C_DIS
LIN {X 51.359,Y 73.646,Z 75.424,A 180.000,B 0.000,C 180.000} C_DIS
LIN {X 51.427,Y 73.685,Z 75.422,A 180.000,B 0.000,C 180.000} C_DIS
LIN {X 51.496,Y 73.722,Z 75.419,A 180.000,B 0.000,C 180.000} C_DIS
LIN {X 51.567,Y 73.757,Z 75.416,A 180.000,B 0.000,C 180.000} C_DIS
LIN {X 51.638,Y 73.790,Z 75.413,A 180.000,B 0.000,C 180.000} C_DIS
LIN {X 51.711,Y 73.820,Z 75.411,A 180.000,B 0.000,C 180.000} C_DIS
LIN {X 51.785,Y 73.849,Z 75.408,A 180.000,B 0.000,C 180.000} C_DIS
LIN {X 51.859,Y 73.874,Z 75.405,A 180.000,B 0.000,C 180.000} C_DIS
LIN {X 51.934,Y 73.898,Z 75.402,A 180.000,B 0.000,C 180.000} C_DIS
LIN {X 52.010,Y 73.919,Z 75.400,A 180.000,B 0.000,C 180.000} C_DIS
LIN {X 52.087,Y 73.938,Z 75.397,A 180.000,B 0.000,C 180.000} C_DIS
LIN {X 52.164,Y 73.954,Z 75.394,A 180.000,B 0.000,C 180.000} C_DIS
LIN {X 52.241,Y 73.968,Z 75.391,A 180.000,B 0.000,C 180.000} C_DIS
LIN {X 52.319,Y 73.979,Z 75.389,A 180.000,B 0.000,C 180.000} C_DIS
LIN {X 52.397,Y 73.988,Z 75.386,A 180.000,B 0.000,C 180.000} C_DIS
LIN {X 52.476,Y 73.995,Z 75.383,A 180.000,B 0.000,C 180.000} C_DIS
LIN {X 52.555,Y 73.998,Z 75.380,A 180.000,B 0.000,C 180.000} C_DIS
LIN {X 52.633,Y 74.000,Z 75.378,A 180.000,B 0.000,C 180.000} C_DIS
LIN {X 52.712,Y 73.999,Z 75.375,A 180.000,B 0.000,C 180.000} C_DIS
LIN {X 52.791,Y 73.996,Z 75.372,A 180.000,B 0.000,C 180.000} C_DIS
LIN {X 52.869,Y 73.990,Z 75.369,A 180.000,B 0.000,C 180.000} C_DIS
LIN {X 52.948,Y 73.981,Z 75.367,A 180.000,B 0.000,C 180.000} C_DIS
LIN {X 53.026,Y 73.970,Z 75.364,A 180.000,B 0.000,C 180.000} C_DIS
LIN {X 53.103,Y 73.957,Z 75.361,A 180.000,B 0.000,C 180.000} C_DIS
LIN {X 53.180,Y 73.941,Z 75.358,A 180.000,B 0.000,C 180.000} C_DIS
LIN {X 53.257,Y 73.923,Z 75.356,A 180.000,B 0.000,C 180.000} C_DIS
LIN {X 53.333,Y 73.902,Z 75.353,A 180.000,B 0.000,C 180.000} C_DIS
LIN {X 53.408,Y 73.879,Z 75.350,A 180.000,B 0.000,C 180.000} C_DIS
LIN {X 53.483,Y 73.854,Z 75.347,A 180.000,B 0.000,C 180.000} C_DIS
LIN {X 53.632,Y 73.804,Z 75.342,A 180.000,B 0.000,C 180.000} C_DIS
LIN {X 54.080,Y 73.653,Z 75.325,A 180.000,B 0.000,C 180.000} C_DIS
LIN {X 54.155,Y 73.628,Z 75.323,A 180.000,B 0.000,C 180.000} C_DIS
LIN {X 54.304,Y 73.578,Z 75.317,A 180.000,B 0.000,C 180.000} C_DIS
LIN {X 54.752,Y 73.427,Z 75.301,A 180.000,B 0.000,C 180.000} C_DIS
LIN {X 54.901,Y 73.376,Z 75.295,A 180.000,B 0.000,C 180.000} C_DIS
LIN {X 55.349,Y 73.225,Z 75.279,A 180.000,B 0.000,C 180.000} C_DIS
LIN {X 55.498,Y 73.175,Z 75.273,A 180.000,B 0.000,C 180.000} C_DIS
LIN {X 55.722,Y 73.099,Z 75.265,A 180.000,B 0.000,C 180.000} C_DIS
LIN {X 55.871,Y 73.049,Z 75.259,A 180.000,B 0.000,C 180.000} C_DIS
LIN {X 55.945,Y 73.024,Z 75.257,A 180.000,B 0.000,C 180.000} C_DIS
LIN {X 56.095,Y 72.973,Z 75.251,A 180.000,B 0.000,C 180.000} C_DIS
LIN {X 56.319,Y 72.898,Z 75.243,A 180.000,B 0.000,C 180.000} C_DIS
LIN {X 56.468,Y 72.848,Z 75.237,A 180.000,B 0.000,C 180.000} C_DIS
LIN {X 56.542,Y 72.822,Z 75.235,A 180.000,B 0.000,C 180.000} C_DIS
LIN {X 56.692,Y 72.772,Z 75.229,A 180.000,B 0.000,C 180.000} C_DIS
LIN {X 56.916,Y 72.697,Z 75.221,A 180.000,B 0.000,C 180.000} C_DIS
LIN {X 57.065,Y 72.646,Z 75.215,A 180.000,B 0.000,C 180.000} C_DIS
LIN {X 57.139,Y 72.621,Z 75.213,A 180.000,B 0.000,C 180.000} C_DIS
LIN {X 57.289,Y 72.571,Z 75.207,A 180.000,B 0.000,C 180.000} C_DIS
LIN {X 57.512,Y 72.495,Z 75.199,A 180.000,B 0.000,C 180.000} C_DIS
LIN {X 57.662,Y 72.445,Z 75.193,A 180.000,B 0.000,C 180.000} C_DIS
LIN {X 57.960,Y 72.344,Z 75.182,A 180.000,B 0.000,C 180.000} C_DIS
LIN {X 58.109,Y 72.294,Z 75.177,A 180.000,B 0.000,C 180.000} C_DIS
LIN {X 58.259,Y 72.243,Z 75.172,A 180.000,B 0.000,C 180.000} C_DIS
LIN {X 58.408,Y 72.193,Z 75.166,A 180.000,B 0.000,C 180.000} C_DIS
LIN {X 58.483,Y 72.168,Z 75.164,A 180.000,B 0.000,C 180.000} C_DIS
LIN {X 58.557,Y 72.143,Z 75.161,A 180.000,B 0.000,C 180.000} C_DIS
LIN {X 58.632,Y 72.118,Z 75.159,A 180.000,B 0.000,C 180.000} C_DIS
LIN {X 58.706,Y 72.092,Z 75.156,A 180.000,B 0.000,C 180.000} C_DIS
LIN {X 58.781,Y 72.067,Z 75.154,A 180.000,B 0.000,C 180.000} C_DIS
LIN {X 58.856,Y 72.042,Z 75.151,A 180.000,B 0.000,C 180.000} C_DIS
LIN {X 58.930,Y 72.017,Z 75.149,A 180.000,B 0.000,C 180.000} C_DIS
LIN {X 59.079,Y 71.967,Z 75.144,A 180.000,B 0.000,C 180.000} C_DIS
LIN {X 59.229,Y 71.916,Z 75.139,A 180.000,B 0.000,C 180.000} C_DIS
LIN {X 59.378,Y 71.866,Z 75.134,A 180.000,B 0.000,C 180.000} C_DIS
LIN {X 59.527,Y 71.815,Z 75.129,A 180.000,B 0.000,C 180.000} C_DIS
LIN {X 59.676,Y 71.765,Z 75.124,A 180.000,B 0.000,C 180.000} C_DIS
LIN {X 59.826,Y 71.715,Z 75.120,A 180.000,B 0.000,C 180.000} C_DIS
LIN {X 59.975,Y 71.664,Z 75.115,A 180.000,B 0.000,C 180.000} C_DIS
LIN {X 60.124,Y 71.614,Z 75.111,A 180.000,B 0.000,C 180.000} C_DIS
LIN {X 60.273,Y 71.564,Z 75.106,A 180.000,B 0.000,C 180.000} C_DIS
LIN {X 60.423,Y 71.513,Z 75.102,A 180.000,B 0.000,C 180.000} C_DIS
LIN {X 60.572,Y 71.463,Z 75.097,A 180.000,B 0.000,C 180.000} C_DIS
LIN {X 60.721,Y 71.413,Z 75.093,A 180.000,B 0.000,C 180.000} C_DIS
LIN {X 60.870,Y 71.362,Z 75.089,A 180.000,B 0.000,C 180.000} C_DIS
LIN {X 61.020,Y 71.312,Z 75.085,A 180.000,B 0.000,C 180.000} C_DIS
LIN {X 61.169,Y 71.262,Z 75.081,A 180.000,B 0.000,C 180.000} C_DIS
LIN {X 61.318,Y 71.211,Z 75.077,A 180.000,B 0.000,C 180.000} C_DIS
LIN {X 61.467,Y 71.161,Z 75.073,A 180.000,B 0.000,C 180.000} C_DIS
LIN {X 61.616,Y 71.111,Z 75.070,A 180.000,B 0.000,C 180.000} C_DIS
LIN {X 61.766,Y 71.060,Z 75.066,A 180.000,B 0.000,C 180.000} C_DIS
LIN {X 61.915,Y 71.010,Z 75.062,A 180.000,B 0.000,C 180.000} C_DIS
LIN {X 62.064,Y 70.960,Z 75.059,A 180.000,B 0.000,C 180.000} C_DIS
LIN {X 62.213,Y 70.909,Z 75.056,A 180.000,B 0.000,C 180.000} C_DIS
LIN {X 62.363,Y 70.859,Z 75.052,A 180.000,B 0.000,C 180.000} C_DIS
LIN {X 62.512,Y 70.809,Z 75.049,A 180.000,B 0.000,C 180.000} C_DIS
LIN {X 62.661,Y 70.758,Z 75.046,A 180.000,B 0.000,C 180.000} C_DIS
LIN {X 62.810,Y 70.708,Z 75.043,A 180.000,B 0.000,C 180.000} C_DIS
LIN {X 62.960,Y 70.658,Z 75.040,A 180.000,B 0.000,C 180.000} C_DIS
LIN {X 63.109,Y 70.607,Z 75.037,A 180.000,B 0.000,C 180.000} C_DIS
LIN {X 63.258,Y 70.557,Z 75.034,A 180.000,B 0.000,C 180.000} C_DIS
LIN {X 63.407,Y 70.507,Z 75.032,A 180.000,B 0.000,C 180.000} C_DIS
LIN {X 63.557,Y 70.456,Z 75.029,A 180.000,B 0.000,C 180.000} C_DIS
LIN {X 63.706,Y 70.406,Z 75.027,A 180.000,B 0.000,C 180.000} C_DIS
LIN {X 64.004,Y 70.305,Z 75.022,A 180.000,B 0.000,C 180.000} C_DIS
LIN {X 64.303,Y 70.204,Z 75.018,A 180.000,B 0.000,C 180.000} C_DIS
LIN {X 64.601,Y 70.104,Z 75.014,A 180.000,B 0.000,C 180.000} C_DIS
LIN {X 64.900,Y 70.003,Z 75.011,A 180.000,B 0.000,C 180.000} C_DIS
LIN {X 65.198,Y 69.902,Z 75.008,A 180.000,B 0.000,C 180.000} C_DIS
LIN {X 65.497,Y 69.802,Z 75.005,A 180.000,B 0.000,C 180.000} C_DIS
LIN {X 65.795,Y 69.701,Z 75.003,A 180.000,B 0.000,C 180.000} C_DIS
LIN {X 66.094,Y 69.600,Z 75.002,A 180.000,B 0.000,C 180.000} C_DIS
LIN {X 66.392,Y 69.500,Z 75.001,A 180.000,B 0.000,C 180.000} C_DIS
LIN {X 66.691,Y 69.399,Z 75.000,A 180.000,B 0.000,C 180.000} C_DIS
LIN {X 66.911,Y 69.325,Z 75.000,A 180.000,B 0.000,C 180.000} C_DIS
; Cutting Move Starts
LIN {X 73.677,Y 67.042,Z 75.000,A 180.000,B 0.000,C 180.000} C_DIS
LIN {X 73.835,Y 66.985,Z 75.000,A 180.000,B 0.000,C 180.000} C_DIS
LIN {X 73.925,Y 66.947,Z 75.000,A 180.000,B 0.000,C 180.000} C_DIS
LIN {X 74.014,Y 66.905,Z 75.000,A 180.000,B 0.000,C 180.000} C_DIS
LIN {X 74.095,Y 66.863,Z 75.000,A 180.000,B 0.000,C 180.000} C_DIS
LIN {X 74.193,Y 66.807,Z 75.000,A 180.000,B 0.000,C 180.000} C_DIS
LIN {X 74.282,Y 66.751,Z 75.000,A 180.000,B 0.000,C 180.000} C_DIS
LIN {X 74.372,Y 66.689,Z 75.000,A 180.000,B 0.000,C 180.000} C_DIS
LIN {X 74.378,Y 66.684,Z 75.000,A 180.000,B 0.000,C 180.000} C_DIS
LIN {X 74.464,Y 66.619,Z 75.000,A 180.000,B 0.000,C 180.000} C_DIS
LIN {X 74.550,Y 66.547,Z 75.000,A 180.000,B 0.000,C 180.000} C_DIS
LIN {X 74.597,Y 66.506,Z 75.000,A 180.000,B 0.000,C 180.000} C_DIS
LIN {X 74.663,Y 66.443,Z 75.000,A 180.000,B 0.000,C 180.000} C_DIS
LIN {X 74.729,Y 66.375,Z 75.000,A 180.000,B 0.000,C 180.000} C_DIS
LIN {X 74.773,Y 66.327,Z 75.000,A 180.000,B 0.000,C 180.000} C_DIS
LIN {X 74.843,Y 66.244,Z 75.000,A 180.000,B 0.000,C 180.000} C_DIS
LIN {X 74.908,Y 66.162,Z 75.000,A 180.000,B 0.000,C 180.000} C_DIS
LIN {X 74.918,Y 66.148,Z 75.000,A 180.000,B 0.000,C 180.000} C_DIS
LIN {X 74.981,Y 66.059,Z 75.000,A 180.000,B 0.000,C 180.000} C_DIS
LIN {X 75.038,Y 65.969,Z 75.000,A 180.000,B 0.000,C 180.000} C_DIS
LIN {X 75.087,Y 65.887,Z 75.000,A 180.000,B 0.000,C 180.000} C_DIS
LIN {X 75.138,Y 65.791,Z 75.000,A 180.000,B 0.000,C 180.000} C_DIS
LIN {X 75.220,Y 65.612,Z 75.000,A 180.000,B 0.000,C 180.000} C_DIS
LIN {X 75.265,Y 65.491,Z 75.000,A 180.000,B 0.000,C 180.000} C_DIS
LIN {X 75.285,Y 65.433,Z 75.000,A 180.000,B 0.000,C 180.000} C_DIS
LIN {X 75.336,Y 65.254,Z 75.000,A 180.000,B 0.000,C 180.000} C_DIS
LIN {X 75.372,Y 65.075,Z 75.000,A 180.000,B 0.000,C 180.000} C_DIS
LIN {X 75.395,Y 64.897,Z 75.000,A 180.000,B 0.000,C 180.000} C_DIS
LIN {X 75.406,Y 64.718,Z 75.000,A 180.000,B 0.000,C 180.000} C_DIS
LIN {X 75.403,Y 64.539,Z 75.000,A 180.000,B 0.000,C 180.000} C_DIS
LIN {X 75.388,Y 64.360,Z 75.000,A 180.000,B 0.000,C 180.000} C_DIS
LIN {X 75.359,Y 64.182,Z 75.000,A 180.000,B 0.000,C 180.000} C_DIS
LIN {X 75.317,Y 64.003,Z 75.000,A 180.000,B 0.000,C 180.000} C_DIS
LIN {X 75.265,Y 63.835,Z 75.000,A 180.000,B 0.000,C 180.000} C_DIS
LIN {X 68.929,Y 45.053,Z 75.000,A 180.000,B 0.000,C 180.000} C_DIS
LIN {X 68.869,Y 44.874,Z 75.000,A 180.000,B 0.000,C 180.000} C_DIS
LIN {X 68.830,Y 44.772,Z 75.000,A 180.000,B 0.000,C 180.000} C_DIS
LIN {X 68.797,Y 44.696,Z 75.000,A 180.000,B 0.000,C 180.000} C_DIS
LIN {X 68.709,Y 44.517,Z 75.000,A 180.000,B 0.000,C 180.000} C_DIS
LIN {X 68.651,Y 44.416,Z 75.000,A 180.000,B 0.000,C 180.000} C_DIS
LIN {X 68.601,Y 44.338,Z 75.000,A 180.000,B 0.000,C 180.000} C_DIS
LIN {X 68.472,Y 44.159,Z 75.000,A 180.000,B 0.000,C 180.000} C_DIS
LIN {X 68.316,Y 43.981,Z 75.000,A 180.000,B 0.000,C 180.000} C_DIS
LIN {X 68.293,Y 43.957,Z 75.000,A 180.000,B 0.000,C 180.000} C_DIS
LIN {X 68.125,Y 43.802,Z 75.000,A 180.000,B 0.000,C 180.000} C_DIS
LIN {X 68.115,Y 43.793,Z 75.000,A 180.000,B 0.000,C 180.000} C_DIS
LIN {X 67.936,Y 43.657,Z 75.000,A 180.000,B 0.000,C 180.000} C_DIS
LIN {X 67.886,Y 43.623,Z 75.000,A 180.000,B 0.000,C 180.000} C_DIS
LIN {X 67.757,Y 43.544,Z 75.000,A 180.000,B 0.000,C 180.000} C_DIS
LIN {X 67.578,Y 43.451,Z 75.000,A 180.000,B 0.000,C 180.000} C_DIS
LIN {X 67.564,Y 43.444,Z 75.000,A 180.000,B 0.000,C 180.000} C_DIS
LIN {X 67.399,Y 43.375,Z 75.000,A 180.000,B 0.000,C 180.000} C_DIS
LIN {X 67.221,Y 43.315,Z 75.000,A 180.000,B 0.000,C 180.000} C_DIS
LIN {X 67.042,Y 43.269,Z 75.000,A 180.000,B 0.000,C 180.000} C_DIS
LIN {X 67.024,Y 43.266,Z 75.000,A 180.000,B 0.000,C 180.000} C_DIS
LIN {X 66.863,Y 43.237,Z 75.000,A 180.000,B 0.000,C 180.000} C_DIS
LIN {X 66.774,Y 43.226,Z 75.000,A 180.000,B 0.000,C 180.000} C_DIS
LIN {X 66.684,Y 43.219,Z 75.000,A 180.000,B 0.000,C 180.000} C_DIS
LIN {X 66.595,Y 43.214,Z 75.000,A 180.000,B 0.000,C 180.000} C_DIS
LIN {X 66.506,Y 43.213,Z 75.000,A 180.000,B 0.000,C 180.000} C_DIS
LIN {X 66.416,Y 43.215,Z 75.000,A 180.000,B 0.000,C 180.000} C_DIS
LIN {X 66.327,Y 43.220,Z 75.000,A 180.000,B 0.000,C 180.000} C_DIS
LIN {X 66.237,Y 43.228,Z 75.000,A 180.000,B 0.000,C 180.000} C_DIS
LIN {X 66.148,Y 43.240,Z 75.000,A 180.000,B 0.000,C 180.000} C_DIS
LIN {X 66.075,Y 43.252,Z 75.000,A 180.000,B 0.000,C 180.000} C_DIS
LIN {X 66.003,Y 43.266,Z 75.000,A 180.000,B 0.000,C 180.000} C_DIS
LIN {X 65.969,Y 43.273,Z 75.000,A 180.000,B 0.000,C 180.000} C_DIS
LIN {X 65.880,Y 43.294,Z 75.000,A 180.000,B 0.000,C 180.000} C_DIS
LIN {X 65.791,Y 43.320,Z 75.000,A 180.000,B 0.000,C 180.000} C_DIS
LIN {X 65.612,Y 43.379,Z 75.000,A 180.000,B 0.000,C 180.000} C_DIS
LIN {X 45.590,Y 50.133,Z 75.000,A 180.000,B 0.000,C 180.000} C_DIS
LIN {X 45.411,Y 50.194,Z 75.000,A 180.000,B 0.000,C 180.000} C_DIS
LIN {X 45.296,Y 50.238,Z 75.000,A 180.000,B 0.000,C 180.000} C_DIS
LIN {X 45.232,Y 50.265,Z 75.000,A 180.000,B 0.000,C 180.000} C_DIS
LIN {X 45.053,Y 50.353,Z 75.000,A 180.000,B 0.000,C 180.000} C_DIS
LIN {X 44.944,Y 50.416,Z 75.000,A 180.000,B 0.000,C 180.000} C_DIS
LIN {X 44.874,Y 50.461,Z 75.000,A 180.000,B 0.000,C 180.000} C_DIS
LIN {X 44.785,Y 50.522,Z 75.000,A 180.000,B 0.000,C 180.000} C_DIS
LIN {X 44.696,Y 50.590,Z 75.000,A 180.000,B 0.000,C 180.000} C_DIS
LIN {X 44.689,Y 50.595,Z 75.000,A 180.000,B 0.000,C 180.000} C_DIS
LIN {X 44.603,Y 50.667,Z 75.000,A 180.000,B 0.000,C 180.000} C_DIS
LIN {X 44.517,Y 50.746,Z 75.000,A 180.000,B 0.000,C 180.000} C_DIS
LIN {X 44.488,Y 50.774,Z 75.000,A 180.000,B 0.000,C 180.000} C_DIS
LIN {X 44.410,Y 50.855,Z 75.000,A 180.000,B 0.000,C 180.000} C_DIS
LIN {X 44.338,Y 50.936,Z 75.000,A 180.000,B 0.000,C 180.000} C_DIS
LIN {X 44.325,Y 50.953,Z 75.000,A 180.000,B 0.000,C 180.000} C_DIS
LIN {X 44.254,Y 51.042,Z 75.000,A 180.000,B 0.000,C 180.000} C_DIS
LIN {X 44.189,Y 51.131,Z 75.000,A 180.000,B 0.000,C 180.000} C_DIS
LIN {X 44.159,Y 51.176,Z 75.000,A 180.000,B 0.000,C 180.000} C_DIS
LIN {X 44.077,Y 51.310,Z 75.000,A 180.000,B 0.000,C 180.000} C_DIS
LIN {X 43.984,Y 51.489,Z 75.000,A 180.000,B 0.000,C 180.000} C_DIS
LIN {X 43.981,Y 51.497,Z 75.000,A 180.000,B 0.000,C 180.000} C_DIS
LIN {X 43.909,Y 51.668,Z 75.000,A 180.000,B 0.000,C 180.000} C_DIS
LIN {X 43.849,Y 51.847,Z 75.000,A 180.000,B 0.000,C 180.000} C_DIS
LIN {X 43.804,Y 52.025,Z 75.000,A 180.000,B 0.000,C 180.000} C_DIS
LIN {X 43.802,Y 52.035,Z 75.000,A 180.000,B 0.000,C 180.000} C_DIS
LIN {X 43.772,Y 52.204,Z 75.000,A 180.000,B 0.000,C 180.000} C_DIS
LIN {X 43.754,Y 52.383,Z 75.000,A 180.000,B 0.000,C 180.000} C_DIS
LIN {X 43.748,Y 52.562,Z 75.000,A 180.000,B 0.000,C 180.000} C_DIS
LIN {X 43.756,Y 52.740,Z 75.000,A 180.000,B 0.000,C 180.000} C_DIS
LIN {X 43.776,Y 52.919,Z 75.000,A 180.000,B 0.000,C 180.000} C_DIS
LIN {X 43.802,Y 53.064,Z 75.000,A 180.000,B 0.000,C 180.000} C_DIS
LIN {X 43.809,Y 53.098,Z 75.000,A 180.000,B 0.000,C 180.000} C_DIS
LIN {X 43.856,Y 53.277,Z 75.000,A 180.000,B 0.000,C 180.000} C_DIS
LIN {X 43.916,Y 53.455,Z 75.000,A 180.000,B 0.000,C 180.000} C_DIS
LIN {X 50.248,Y 72.226,Z 75.000,A 180.000,B 0.000,C 180.000} C_DIS
LIN {X 50.311,Y 72.405,Z 75.000,A 180.000,B 0.000,C 180.000} C_DIS
LIN {X 50.388,Y 72.584,Z 75.000,A 180.000,B 0.000,C 180.000} C_DIS
LIN {X 50.416,Y 72.640,Z 75.000,A 180.000,B 0.000,C 180.000} C_DIS
LIN {X 50.484,Y 72.763,Z 75.000,A 180.000,B 0.000,C 180.000} C_DIS
LIN {X 50.595,Y 72.936,Z 75.000,A 180.000,B 0.000,C 180.000} C_DIS
LIN {X 50.599,Y 72.941,Z 75.000,A 180.000,B 0.000,C 180.000} C_DIS
LIN {X 50.665,Y 73.031,Z 75.000,A 180.000,B 0.000,C 180.000} C_DIS
LIN {X 50.737,Y 73.120,Z 75.000,A 180.000,B 0.000,C 180.000} C_DIS
LIN {X 50.774,Y 73.162,Z 75.000,A 180.000,B 0.000,C 180.000} C_DIS
LIN {X 50.905,Y 73.299,Z 75.000,A 180.000,B 0.000,C 180.000} C_DIS
LIN {X 50.953,Y 73.343,Z 75.000,A 180.000,B 0.000,C 180.000} C_DIS
LIN {X 51.112,Y 73.478,Z 75.000,A 180.000,B 0.000,C 180.000} C_DIS
LIN {X 51.131,Y 73.493,Z 75.000,A 180.000,B 0.000,C 180.000} C_DIS
LIN {X 51.310,Y 73.616,Z 75.000,A 180.000,B 0.000,C 180.000} C_DIS
LIN {X 51.376,Y 73.656,Z 75.000,A 180.000,B 0.000,C 180.000} C_DIS
LIN {X 51.489,Y 73.719,Z 75.000,A 180.000,B 0.000,C 180.000} C_DIS
LIN {X 51.668,Y 73.803,Z 75.000,A 180.000,B 0.000,C 180.000} C_DIS
LIN {X 51.749,Y 73.835,Z 75.000,A 180.000,B 0.000,C 180.000} C_DIS
LIN {X 51.847,Y 73.870,Z 75.000,A 180.000,B 0.000,C 180.000} C_DIS
LIN {X 52.025,Y 73.923,Z 75.000,A 180.000,B 0.000,C 180.000} C_DIS
LIN {X 52.204,Y 73.961,Z 75.000,A 180.000,B 0.000,C 180.000} C_DIS
LIN {X 52.383,Y 73.987,Z 75.000,A 180.000,B 0.000,C 180.000} C_DIS
LIN {X 52.562,Y 73.999,Z 75.000,A 180.000,B 0.000,C 180.000} C_DIS
LIN {X 52.740,Y 73.998,Z 75.000,A 180.000,B 0.000,C 180.000} C_DIS
LIN {X 52.919,Y 73.985,Z 75.000,A 180.000,B 0.000,C 180.000} C_DIS
LIN {X 53.098,Y 73.958,Z 75.000,A 180.000,B 0.000,C 180.000} C_DIS
LIN {X 53.277,Y 73.918,Z 75.000,A 180.000,B 0.000,C 180.000} C_DIS
LIN {X 53.455,Y 73.864,Z 75.000,A 180.000,B 0.000,C 180.000} C_DIS
LIN {X 66.911,Y 69.325,Z 75.000,A 180.000,B 0.000,C 180.000} C_DIS
; Link Move Starts
LIN {X 67.209,Y 69.224,Z 75.000,A 180.000,B 0.000,C 180.000} C_DIS
LIN {X 67.508,Y 69.123,Z 74.998,A 180.000,B 0.000,C 180.000} C_DIS
LIN {X 67.806,Y 69.022,Z 74.996,A 180.000,B 0.000,C 180.000} C_DIS
LIN {X 68.105,Y 68.922,Z 74.992,A 180.000,B 0.000,C 180.000} C_DIS
LIN {X 68.403,Y 68.821,Z 74.988,A 180.000,B 0.000,C 180.000} C_DIS
LIN {X 68.702,Y 68.720,Z 74.983,A 180.000,B 0.000,C 180.000} C_DIS
LIN {X 68.851,Y 68.670,Z 74.981,A 180.000,B 0.000,C 180.000} C_DIS
LIN {X 69.000,Y 68.620,Z 74.978,A 180.000,B 0.000,C 180.000} C_DIS
LIN {X 69.150,Y 68.569,Z 74.975,A 180.000,B 0.000,C 180.000} C_DIS
LIN {X 69.299,Y 68.519,Z 74.971,A 180.000,B 0.000,C 180.000} C_DIS
LIN {X 69.448,Y 68.469,Z 74.968,A 180.000,B 0.000,C 180.000} C_DIS
LIN {X 69.597,Y 68.418,Z 74.964,A 180.000,B 0.000,C 180.000} C_DIS
LIN {X 69.746,Y 68.368,Z 74.960,A 180.000,B 0.000,C 180.000} C_DIS
LIN {X 69.896,Y 68.318,Z 74.956,A 180.000,B 0.000,C 180.000} C_DIS
LIN {X 70.045,Y 68.267,Z 74.952,A 180.000,B 0.000,C 180.000} C_DIS
LIN {X 70.194,Y 68.217,Z 74.948,A 180.000,B 0.000,C 180.000} C_DIS
LIN {X 70.343,Y 68.167,Z 74.944,A 180.000,B 0.000,C 180.000} C_DIS
LIN {X 70.493,Y 68.116,Z 74.939,A 180.000,B 0.000,C 180.000} C_DIS
LIN {X 70.642,Y 68.066,Z 74.934,A 180.000,B 0.000,C 180.000} C_DIS
LIN {X 70.791,Y 68.016,Z 74.929,A 180.000,B 0.000,C 180.000} C_DIS
LIN {X 70.940,Y 67.965,Z 74.924,A 180.000,B 0.000,C 180.000} C_DIS
LIN {X 71.015,Y 67.940,Z 74.922,A 180.000,B 0.000,C 180.000} C_DIS
LIN {X 71.090,Y 67.915,Z 74.919,A 180.000,B 0.000,C 180.000} C_DIS
LIN {X 71.164,Y 67.890,Z 74.917,A 180.000,B 0.000,C 180.000} C_DIS
LIN {X 71.239,Y 67.865,Z 74.914,A 180.000,B 0.000,C 180.000} C_DIS
LIN {X 71.313,Y 67.839,Z 74.911,A 180.000,B 0.000,C 180.000} C_DIS
LIN {X 71.388,Y 67.814,Z 74.909,A 180.000,B 0.000,C 180.000} C_DIS
LIN {X 71.463,Y 67.789,Z 74.906,A 180.000,B 0.000,C 180.000} C_DIS
LIN {X 71.537,Y 67.764,Z 74.903,A 180.000,B 0.000,C 180.000} C_DIS
LIN {X 71.612,Y 67.739,Z 74.901,A 180.000,B 0.000,C 180.000} C_DIS
LIN {X 71.687,Y 67.714,Z 74.898,A 180.000,B 0.000,C 180.000} C_DIS
LIN {X 71.761,Y 67.688,Z 74.895,A 180.000,B 0.000,C 180.000} C_DIS
LIN {X 71.836,Y 67.663,Z 74.892,A 180.000,B 0.000,C 180.000} C_DIS
LIN {X 71.910,Y 67.638,Z 74.890,A 180.000,B 0.000,C 180.000} C_DIS
LIN {X 71.985,Y 67.613,Z 74.887,A 180.000,B 0.000,C 180.000} C_DIS
LIN {X 72.060,Y 67.588,Z 74.884,A 180.000,B 0.000,C 180.000} C_DIS
LIN {X 72.134,Y 67.562,Z 74.881,A 180.000,B 0.000,C 180.000} C_DIS
LIN {X 72.209,Y 67.537,Z 74.878,A 180.000,B 0.000,C 180.000} C_DIS
LIN {X 72.283,Y 67.512,Z 74.876,A 180.000,B 0.000,C 180.000} C_DIS
LIN {X 72.358,Y 67.487,Z 74.873,A 180.000,B 0.000,C 180.000} C_DIS
LIN {X 72.433,Y 67.462,Z 74.870,A 180.000,B 0.000,C 180.000} C_DIS
LIN {X 72.507,Y 67.437,Z 74.867,A 180.000,B 0.000,C 180.000} C_DIS
LIN {X 72.582,Y 67.411,Z 74.865,A 180.000,B 0.000,C 180.000} C_DIS
LIN {X 72.657,Y 67.386,Z 74.862,A 180.000,B 0.000,C 180.000} C_DIS
LIN {X 72.806,Y 67.336,Z 74.856,A 180.000,B 0.000,C 180.000} C_DIS
LIN {X 72.880,Y 67.311,Z 74.854,A 180.000,B 0.000,C 180.000} C_DIS
LIN {X 73.030,Y 67.260,Z 74.848,A 180.000,B 0.000,C 180.000} C_DIS
LIN {X 73.254,Y 67.185,Z 74.840,A 180.000,B 0.000,C 180.000} C_DIS
LIN {X 73.403,Y 67.135,Z 74.834,A 180.000,B 0.000,C 180.000} C_DIS
LIN {X 73.477,Y 67.109,Z 74.832,A 180.000,B 0.000,C 180.000} C_DIS
LIN {X 73.627,Y 67.059,Z 74.826,A 180.000,B 0.000,C 180.000} C_DIS
LIN {X 73.851,Y 66.984,Z 74.818,A 180.000,B 0.000,C 180.000} C_DIS
LIN {X 73.925,Y 66.958,Z 74.815,A 180.000,B 0.000,C 180.000} C_DIS
LIN {X 73.999,Y 66.932,Z 74.812,A 180.000,B 0.000,C 180.000} C_DIS
LIN {X 74.073,Y 66.903,Z 74.810,A 180.000,B 0.000,C 180.000} C_DIS
LIN {X 74.145,Y 66.872,Z 74.807,A 180.000,B 0.000,C 180.000} C_DIS
LIN {X 74.217,Y 66.839,Z 74.804,A 180.000,B 0.000,C 180.000} C_DIS
LIN {X 74.288,Y 66.804,Z 74.801,A 180.000,B 0.000,C 180.000} C_DIS
LIN {X 74.357,Y 66.767,Z 74.799,A 180.000,B 0.000,C 180.000} C_DIS
LIN {X 74.425,Y 66.729,Z 74.796,A 180.000,B 0.000,C 180.000} C_DIS
LIN {X 74.491,Y 66.689,Z 74.793,A 180.000,B 0.000,C 180.000} C_DIS
LIN {X 74.555,Y 66.647,Z 74.791,A 180.000,B 0.000,C 180.000} C_DIS
LIN {X 74.619,Y 66.603,Z 74.788,A 180.000,B 0.000,C 180.000} C_DIS
LIN {X 74.681,Y 66.558,Z 74.785,A 180.000,B 0.000,C 180.000} C_DIS
LIN {X 74.741,Y 66.512,Z 74.783,A 180.000,B 0.000,C 180.000} C_DIS
LIN {X 74.800,Y 66.463,Z 74.780,A 180.000,B 0.000,C 180.000} C_DIS
LIN {X 74.858,Y 66.413,Z 74.777,A 180.000,B 0.000,C 180.000} C_DIS
LIN {X 74.912,Y 66.363,Z 74.775,A 180.000,B 0.000,C 180.000} C_DIS
LIN {X 74.966,Y 66.311,Z 74.772,A 180.000,B 0.000,C 180.000} C_DIS
LIN {X 75.018,Y 66.258,Z 74.769,A 180.000,B 0.000,C 180.000} C_DIS
LIN {X 75.068,Y 66.203,Z 74.767,A 180.000,B 0.000,C 180.000} C_DIS
LIN {X 75.117,Y 66.147,Z 74.764,A 180.000,B 0.000,C 180.000} C_DIS
LIN {X 75.165,Y 66.089,Z 74.762,A 180.000,B 0.000,C 180.000} C_DIS
LIN {X 75.211,Y 66.030,Z 74.759,A 180.000,B 0.000,C 180.000} C_DIS
LIN {X 75.255,Y 65.970,Z 74.756,A 180.000,B 0.000,C 180.000} C_DIS
LIN {X 75.297,Y 65.909,Z 74.754,A 180.000,B 0.000,C 180.000} C_DIS
LIN {X 75.337,Y 65.848,Z 74.751,A 180.000,B 0.000,C 180.000} C_DIS
LIN {X 75.375,Y 65.785,Z 74.749,A 180.000,B 0.000,C 180.000} C_DIS
LIN {X 75.412,Y 65.722,Z 74.746,A 180.000,B 0.000,C 180.000} C_DIS
LIN {X 75.446,Y 65.659,Z 74.744,A 180.000,B 0.000,C 180.000} C_DIS
LIN {X 75.479,Y 65.595,Z 74.741,A 180.000,B 0.000,C 180.000} C_DIS
LIN {X 75.509,Y 65.530,Z 74.739,A 180.000,B 0.000,C 180.000} C_DIS
LIN {X 75.538,Y 65.464,Z 74.736,A 180.000,B 0.000,C 180.000} C_DIS
LIN {X 75.566,Y 65.397,Z 74.734,A 180.000,B 0.000,C 180.000} C_DIS
LIN {X 75.592,Y 65.328,Z 74.731,A 180.000,B 0.000,C 180.000} C_DIS
LIN {X 75.615,Y 65.260,Z 74.729,A 180.000,B 0.000,C 180.000} C_DIS
LIN {X 75.637,Y 65.190,Z 74.726,A 180.000,B 0.000,C 180.000} C_DIS
LIN {X 75.657,Y 65.120,Z 74.723,A 180.000,B 0.000,C 180.000} C_DIS
LIN {X 75.675,Y 65.050,Z 74.721,A 180.000,B 0.000,C 180.000} C_DIS
LIN {X 75.691,Y 64.979,Z 74.718,A 180.000,B 0.000,C 180.000} C_DIS
LIN {X 75.705,Y 64.908,Z 74.716,A 180.000,B 0.000,C 180.000} C_DIS
LIN {X 75.726,Y 64.769,Z 74.711,A 180.000,B 0.000,C 180.000} C_DIS
LIN {X 75.740,Y 64.628,Z 74.706,A 180.000,B 0.000,C 180.000} C_DIS
LIN {X 75.746,Y 64.487,Z 74.701,A 180.000,B 0.000,C 180.000} C_DIS
LIN {X 75.744,Y 64.345,Z 74.696,A 180.000,B 0.000,C 180.000} C_DIS
LIN {X 75.740,Y 64.271,Z 74.694,A 180.000,B 0.000,C 180.000} C_DIS
LIN {X 75.734,Y 64.198,Z 74.691,A 180.000,B 0.000,C 180.000} C_DIS
LIN {X 75.726,Y 64.124,Z 74.688,A 180.000,B 0.000,C 180.000} C_DIS
LIN {X 75.715,Y 64.051,Z 74.686,A 180.000,B 0.000,C 180.000} C_DIS
LIN {X 75.703,Y 63.980,Z 74.683,A 180.000,B 0.000,C 180.000} C_DIS
LIN {X 75.689,Y 63.909,Z 74.681,A 180.000,B 0.000,C 180.000} C_DIS
LIN {X 75.672,Y 63.839,Z 74.678,A 180.000,B 0.000,C 180.000} C_DIS
LIN {X 75.654,Y 63.770,Z 74.676,A 180.000,B 0.000,C 180.000} C_DIS
LIN {X 75.633,Y 63.695,Z 74.673,A 180.000,B 0.000,C 180.000} C_DIS
LIN {X 75.589,Y 63.547,Z 74.668,A 180.000,B 0.000,C 180.000} C_DIS
LIN {X 75.568,Y 63.472,Z 74.665,A 180.000,B 0.000,C 180.000} C_DIS
LIN {X 75.546,Y 63.396,Z 74.662,A 180.000,B 0.000,C 180.000} C_DIS
LIN {X 75.524,Y 63.321,Z 74.659,A 180.000,B 0.000,C 180.000} C_DIS
LIN {X 75.502,Y 63.245,Z 74.657,A 180.000,B 0.000,C 180.000} C_DIS
LIN {X 75.479,Y 63.169,Z 74.654,A 180.000,B 0.000,C 180.000} C_DIS
LIN {X 75.457,Y 63.094,Z 74.651,A 180.000,B 0.000,C 180.000} C_DIS
LIN {X 75.435,Y 63.018,Z 74.648,A 180.000,B 0.000,C 180.000} C_DIS
LIN {X 75.413,Y 62.942,Z 74.646,A 180.000,B 0.000,C 180.000} C_DIS
LIN {X 75.391,Y 62.867,Z 74.643,A 180.000,B 0.000,C 180.000} C_DIS
LIN {X 75.369,Y 62.791,Z 74.640,A 180.000,B 0.000,C 180.000} C_DIS
LIN {X 75.347,Y 62.715,Z 74.637,A 180.000,B 0.000,C 180.000} C_DIS
LIN {X 75.325,Y 62.640,Z 74.635,A 180.000,B 0.000,C 180.000} C_DIS
LIN {X 75.303,Y 62.564,Z 74.632,A 180.000,B 0.000,C 180.000} C_DIS
LIN {X 75.281,Y 62.488,Z 74.629,A 180.000,B 0.000,C 180.000} C_DIS
LIN {X 75.259,Y 62.413,Z 74.626,A 180.000,B 0.000,C 180.000} C_DIS
LIN {X 75.237,Y 62.337,Z 74.624,A 180.000,B 0.000,C 180.000} C_DIS
LIN {X 75.215,Y 62.261,Z 74.621,A 180.000,B 0.000,C 180.000} C_DIS
LIN {X 75.193,Y 62.186,Z 74.618,A 180.000,B 0.000,C 180.000} C_DIS
LIN {X 75.171,Y 62.110,Z 74.615,A 180.000,B 0.000,C 180.000} C_DIS
LIN {X 75.149,Y 62.034,Z 74.613,A 180.000,B 0.000,C 180.000} C_DIS
LIN {X 75.127,Y 61.959,Z 74.610,A 180.000,B 0.000,C 180.000} C_DIS
LIN {X 75.105,Y 61.883,Z 74.607,A 180.000,B 0.000,C 180.000} C_DIS
LIN {X 75.083,Y 61.807,Z 74.604,A 180.000,B 0.000,C 180.000} C_DIS
LIN {X 75.061,Y 61.732,Z 74.602,A 180.000,B 0.000,C 180.000} C_DIS
LIN {X 75.039,Y 61.656,Z 74.599,A 180.000,B 0.000,C 180.000} C_DIS
LIN {X 75.017,Y 61.580,Z 74.596,A 180.000,B 0.000,C 180.000} C_DIS
LIN {X 74.995,Y 61.505,Z 74.593,A 180.000,B 0.000,C 180.000} C_DIS
LIN {X 74.973,Y 61.429,Z 74.591,A 180.000,B 0.000,C 180.000} C_DIS
LIN {X 74.950,Y 61.353,Z 74.588,A 180.000,B 0.000,C 180.000} C_DIS
LIN {X 74.928,Y 61.278,Z 74.585,A 180.000,B 0.000,C 180.000} C_DIS
LIN {X 74.906,Y 61.202,Z 74.583,A 180.000,B 0.000,C 180.000} C_DIS
LIN {X 74.884,Y 61.126,Z 74.580,A 180.000,B 0.000,C 180.000} C_DIS
LIN {X 74.862,Y 61.051,Z 74.578,A 180.000,B 0.000,C 180.000} C_DIS
LIN {X 74.839,Y 60.975,Z 74.575,A 180.000,B 0.000,C 180.000} C_DIS
LIN {X 74.817,Y 60.900,Z 74.572,A 180.000,B 0.000,C 180.000} C_DIS
LIN {X 74.772,Y 60.749,Z 74.568,A 180.000,B 0.000,C 180.000} C_DIS
LIN {X 74.727,Y 60.597,Z 74.563,A 180.000,B 0.000,C 180.000} C_DIS
LIN {X 74.682,Y 60.446,Z 74.558,A 180.000,B 0.000,C 180.000} C_DIS
LIN {X 74.637,Y 60.295,Z 74.554,A 180.000,B 0.000,C 180.000} C_DIS
LIN {X 74.592,Y 60.145,Z 74.549,A 180.000,B 0.000,C 180.000} C_DIS
LIN {X 74.546,Y 59.994,Z 74.545,A 180.000,B 0.000,C 180.000} C_DIS
LIN {X 74.500,Y 59.843,Z 74.541,A 180.000,B 0.000,C 180.000} C_DIS
LIN {X 74.454,Y 59.692,Z 74.537,A 180.000,B 0.000,C 180.000} C_DIS
LIN {X 74.408,Y 59.542,Z 74.534,A 180.000,B 0.000,C 180.000} C_DIS
LIN {X 74.362,Y 59.391,Z 74.530,A 180.000,B 0.000,C 180.000} C_DIS
LIN {X 74.315,Y 59.240,Z 74.527,A 180.000,B 0.000,C 180.000} C_DIS
LIN {X 74.269,Y 59.090,Z 74.523,A 180.000,B 0.000,C 180.000} C_DIS
LIN {X 74.222,Y 58.940,Z 74.520,A 180.000,B 0.000,C 180.000} C_DIS
LIN {X 74.175,Y 58.789,Z 74.518,A 180.000,B 0.000,C 180.000} C_DIS
LIN {X 74.127,Y 58.639,Z 74.515,A 180.000,B 0.000,C 180.000} C_DIS
LIN {X 74.032,Y 58.339,Z 74.510,A 180.000,B 0.000,C 180.000} C_DIS
LIN {X 73.936,Y 58.039,Z 74.506,A 180.000,B 0.000,C 180.000} C_DIS
LIN {X 73.838,Y 57.739,Z 74.503,A 180.000,B 0.000,C 180.000} C_DIS
LIN {X 73.740,Y 57.440,Z 74.501,A 180.000,B 0.000,C 180.000} C_DIS
LIN {X 73.641,Y 57.141,Z 74.500,A 180.000,B 0.000,C 180.000} C_DIS
LIN {X 73.566,Y 56.936,Z 74.500,A 180.000,B 0.000,C 180.000} C_DIS
; Cutting Move Starts
LIN {X 69.496,Y 44.874,Z 74.500,A 180.000,B 0.000,C 180.000} C_DIS
LIN {X 69.436,Y 44.696,Z 74.500,A 180.000,B 0.000,C 180.000} C_DIS
LIN {X 69.366,Y 44.518,Z 74.500,A 180.000,B 0.000,C 180.000} C_DIS
LIN {X 69.365,Y 44.517,Z 74.500,A 180.000,B 0.000,C 180.000} C_DIS
LIN {X 69.278,Y 44.338,Z 74.500,A 180.000,B 0.000,C 180.000} C_DIS
LIN {X 69.187,Y 44.183,Z 74.500,A 180.000,B 0.000,C 180.000} C_DIS
LIN {X 69.172,Y 44.159,Z 74.500,A 180.000,B 0.000,C 180.000} C_DIS
LIN {X 69.044,Y 43.981,Z 74.500,A 180.000,B 0.000,C 180.000} C_DIS
LIN {X 69.008,Y 43.936,Z 74.500,A 180.000,B 0.000,C 180.000} C_DIS
LIN {X 68.890,Y 43.802,Z 74.500,A 180.000,B 0.000,C 180.000} C_DIS
LIN {X 68.830,Y 43.740,Z 74.500,A 180.000,B 0.000,C 180.000} C_DIS
LIN {X 68.702,Y 43.623,Z 74.500,A 180.000,B 0.000,C 180.000} C_DIS
LIN {X 68.651,Y 43.581,Z 74.500,A 180.000,B 0.000,C 180.000} C_DIS
LIN {X 68.472,Y 43.448,Z 74.500,A 180.000,B 0.000,C 180.000} C_DIS
LIN {X 68.466,Y 43.444,Z 74.500,A 180.000,B 0.000,C 180.000} C_DIS
LIN {X 68.293,Y 43.339,Z 74.500,A 180.000,B 0.000,C 180.000} C_DIS
LIN {X 68.151,Y 43.266,Z 74.500,A 180.000,B 0.000,C 180.000} C_DIS
LIN {X 68.115,Y 43.248,Z 74.500,A 180.000,B 0.000,C 180.000} C_DIS
LIN {X 67.936,Y 43.175,Z 74.500,A 180.000,B 0.000,C 180.000} C_DIS
LIN {X 67.757,Y 43.117,Z 74.500,A 180.000,B 0.000,C 180.000} C_DIS
LIN {X 67.639,Y 43.087,Z 74.500,A 180.000,B 0.000,C 180.000} C_DIS
LIN {X 67.578,Y 43.074,Z 74.500,A 180.000,B 0.000,C 180.000} C_DIS
LIN {X 67.399,Y 43.044,Z 74.500,A 180.000,B 0.000,C 180.000} C_DIS
LIN {X 67.310,Y 43.034,Z 74.500,A 180.000,B 0.000,C 180.000} C_DIS
LIN {X 67.221,Y 43.027,Z 74.500,A 180.000,B 0.000,C 180.000} C_DIS
LIN {X 67.131,Y 43.023,Z 74.500,A 180.000,B 0.000,C 180.000} C_DIS
LIN {X 67.042,Y 43.023,Z 74.500,A 180.000,B 0.000,C 180.000} C_DIS
LIN {X 66.953,Y 43.026,Z 74.500,A 180.000,B 0.000,C 180.000} C_DIS
LIN {X 66.863,Y 43.032,Z 74.500,A 180.000,B 0.000,C 180.000} C_DIS
LIN {X 66.774,Y 43.041,Z 74.500,A 180.000,B 0.000,C 180.000} C_DIS
LIN {X 66.684,Y 43.054,Z 74.500,A 180.000,B 0.000,C 180.000} C_DIS
LIN {X 66.600,Y 43.069,Z 74.500,A 180.000,B 0.000,C 180.000} C_DIS
LIN {X 66.515,Y 43.087,Z 74.500,A 180.000,B 0.000,C 180.000} C_DIS
LIN {X 66.506,Y 43.089,Z 74.500,A 180.000,B 0.000,C 180.000} C_DIS
LIN {X 66.416,Y 43.112,Z 74.500,A 180.000,B 0.000,C 180.000} C_DIS
LIN {X 66.327,Y 43.138,Z 74.500,A 180.000,B 0.000,C 180.000} C_DIS
LIN {X 66.148,Y 43.198,Z 74.500,A 180.000,B 0.000,C 180.000} C_DIS
LIN {X 45.590,Y 50.133,Z 74.500,A 180.000,B 0.000,C 180.000} C_DIS
LIN {X 45.411,Y 50.194,Z 74.500,A 180.000,B 0.000,C 180.000} C_DIS
LIN {X 45.296,Y 50.238,Z 74.500,A 180.000,B 0.000,C 180.000} C_DIS
LIN {X 45.232,Y 50.265,Z 74.500,A 180.000,B 0.000,C 180.000} C_DIS
LIN {X 45.053,Y 50.353,Z 74.500,A 180.000,B 0.000,C 180.000} C_DIS
LIN {X 44.944,Y 50.416,Z 74.500,A 180.000,B 0.000,C 180.000} C_DIS
LIN {X 44.874,Y 50.461,Z 74.500,A 180.000,B 0.000,C 180.000} C_DIS
LIN {X 44.785,Y 50.522,Z 74.500,A 180.000,B 0.000,C 180.000} C_DIS
LIN {X 44.696,Y 50.590,Z 74.500,A 180.000,B 0.000,C 180.000} C_DIS
LIN {X 44.689,Y 50.595,Z 74.500,A 180.000,B 0.000,C 180.000} C_DIS
LIN {X 44.603,Y 50.667,Z 74.500,A 180.000,B 0.000,C 180.000} C_DIS
LIN {X 44.517,Y 50.746,Z 74.500,A 180.000,B 0.000,C 180.000} C_DIS
LIN {X 44.488,Y 50.774,Z 74.500,A 180.000,B 0.000,C 180.000} C_DIS
LIN {X 44.410,Y 50.855,Z 74.500,A 180.000,B 0.000,C 180.000} C_DIS
LIN {X 44.338,Y 50.936,Z 74.500,A 180.000,B 0.000,C 180.000} C_DIS
LIN {X 44.325,Y 50.953,Z 74.500,A 180.000,B 0.000,C 180.000} C_DIS
LIN {X 44.254,Y 51.042,Z 74.500,A 180.000,B 0.000,C 180.000} C_DIS
LIN {X 44.189,Y 51.131,Z 74.500,A 180.000,B 0.000,C 180.000} C_DIS
LIN {X 44.159,Y 51.176,Z 74.500,A 180.000,B 0.000,C 180.000} C_DIS
LIN {X 44.077,Y 51.310,Z 74.500,A 180.000,B 0.000,C 180.000} C_DIS
LIN {X 43.984,Y 51.489,Z 74.500,A 180.000,B 0.000,C 180.000} C_DIS
LIN {X 43.981,Y 51.497,Z 74.500,A 180.000,B 0.000,C 180.000} C_DIS
LIN {X 43.909,Y 51.668,Z 74.500,A 180.000,B 0.000,C 180.000} C_DIS
LIN {X 43.849,Y 51.847,Z 74.500,A 180.000,B 0.000,C 180.000} C_DIS
LIN {X 43.804,Y 52.025,Z 74.500,A 180.000,B 0.000,C 180.000} C_DIS
LIN {X 43.802,Y 52.035,Z 74.500,A 180.000,B 0.000,C 180.000} C_DIS
LIN {X 43.772,Y 52.204,Z 74.500,A 180.000,B 0.000,C 180.000} C_DIS
LIN {X 43.754,Y 52.383,Z 74.500,A 180.000,B 0.000,C 180.000} C_DIS
LIN {X 43.748,Y 52.562,Z 74.500,A 180.000,B 0.000,C 180.000} C_DIS
LIN {X 43.756,Y 52.740,Z 74.500,A 180.000,B 0.000,C 180.000} C_DIS
LIN {X 43.776,Y 52.919,Z 74.500,A 180.000,B 0.000,C 180.000} C_DIS
LIN {X 43.802,Y 53.064,Z 74.500,A 180.000,B 0.000,C 180.000} C_DIS
LIN {X 43.809,Y 53.098,Z 74.500,A 180.000,B 0.000,C 180.000} C_DIS
LIN {X 43.856,Y 53.277,Z 74.500,A 180.000,B 0.000,C 180.000} C_DIS
LIN {X 43.916,Y 53.455,Z 74.500,A 180.000,B 0.000,C 180.000} C_DIS
LIN {X 50.248,Y 72.226,Z 74.500,A 180.000,B 0.000,C 180.000} C_DIS
LIN {X 50.311,Y 72.405,Z 74.500,A 180.000,B 0.000,C 180.000} C_DIS
LIN {X 50.388,Y 72.584,Z 74.500,A 180.000,B 0.000,C 180.000} C_DIS
LIN {X 50.416,Y 72.640,Z 74.500,A 180.000,B 0.000,C 180.000} C_DIS
LIN {X 50.484,Y 72.763,Z 74.500,A 180.000,B 0.000,C 180.000} C_DIS
LIN {X 50.595,Y 72.936,Z 74.500,A 180.000,B 0.000,C 180.000} C_DIS
LIN {X 50.599,Y 72.941,Z 74.500,A 180.000,B 0.000,C 180.000} C_DIS
LIN {X 50.665,Y 73.031,Z 74.500,A 180.000,B 0.000,C 180.000} C_DIS
LIN {X 50.737,Y 73.120,Z 74.500,A 180.000,B 0.000,C 180.000} C_DIS
LIN {X 50.774,Y 73.162,Z 74.500,A 180.000,B 0.000,C 180.000} C_DIS
LIN {X 50.905,Y 73.299,Z 74.500,A 180.000,B 0.000,C 180.000} C_DIS
LIN {X 50.953,Y 73.343,Z 74.500,A 180.000,B 0.000,C 180.000} C_DIS
LIN {X 51.112,Y 73.478,Z 74.500,A 180.000,B 0.000,C 180.000} C_DIS
LIN {X 51.131,Y 73.493,Z 74.500,A 180.000,B 0.000,C 180.000} C_DIS
LIN {X 51.310,Y 73.616,Z 74.500,A 180.000,B 0.000,C 180.000} C_DIS
LIN {X 51.376,Y 73.656,Z 74.500,A 180.000,B 0.000,C 180.000} C_DIS
LIN {X 51.489,Y 73.719,Z 74.500,A 180.000,B 0.000,C 180.000} C_DIS
LIN {X 51.668,Y 73.803,Z 74.500,A 180.000,B 0.000,C 180.000} C_DIS
LIN {X 51.749,Y 73.835,Z 74.500,A 180.000,B 0.000,C 180.000} C_DIS
LIN {X 51.847,Y 73.870,Z 74.500,A 180.000,B 0.000,C 180.000} C_DIS
LIN {X 52.025,Y 73.923,Z 74.500,A 180.000,B 0.000,C 180.000} C_DIS
LIN {X 52.204,Y 73.961,Z 74.500,A 180.000,B 0.000,C 180.000} C_DIS
LIN {X 52.383,Y 73.987,Z 74.500,A 180.000,B 0.000,C 180.000} C_DIS
LIN {X 52.562,Y 73.999,Z 74.500,A 180.000,B 0.000,C 180.000} C_DIS
LIN {X 52.740,Y 73.998,Z 74.500,A 180.000,B 0.000,C 180.000} C_DIS
LIN {X 52.919,Y 73.985,Z 74.500,A 180.000,B 0.000,C 180.000} C_DIS
LIN {X 53.098,Y 73.958,Z 74.500,A 180.000,B 0.000,C 180.000} C_DIS
LIN {X 53.277,Y 73.918,Z 74.500,A 180.000,B 0.000,C 180.000} C_DIS
LIN {X 53.455,Y 73.864,Z 74.500,A 180.000,B 0.000,C 180.000} C_DIS
LIN {X 74.207,Y 66.863,Z 74.500,A 180.000,B 0.000,C 180.000} C_DIS
LIN {X 74.372,Y 66.805,Z 74.500,A 180.000,B 0.000,C 180.000} C_DIS
LIN {X 74.461,Y 66.769,Z 74.500,A 180.000,B 0.000,C 180.000} C_DIS
LIN {X 74.550,Y 66.728,Z 74.500,A 180.000,B 0.000,C 180.000} C_DIS
LIN {X 74.637,Y 66.684,Z 74.500,A 180.000,B 0.000,C 180.000} C_DIS
LIN {X 74.729,Y 66.633,Z 74.500,A 180.000,B 0.000,C 180.000} C_DIS
LIN {X 74.818,Y 66.579,Z 74.500,A 180.000,B 0.000,C 180.000} C_DIS
LIN {X 74.908,Y 66.519,Z 74.500,A 180.000,B 0.000,C 180.000} C_DIS
LIN {X 74.926,Y 66.506,Z 74.500,A 180.000,B 0.000,C 180.000} C_DIS
LIN {X 75.006,Y 66.446,Z 74.500,A 180.000,B 0.000,C 180.000} C_DIS
LIN {X 75.087,Y 66.380,Z 74.500,A 180.000,B 0.000,C 180.000} C_DIS
LIN {X 75.148,Y 66.327,Z 74.500,A 180.000,B 0.000,C 180.000} C_DIS
LIN {X 75.265,Y 66.213,Z 74.500,A 180.000,B 0.000,C 180.000} C_DIS
LIN {X 75.326,Y 66.148,Z 74.500,A 180.000,B 0.000,C 180.000} C_DIS
LIN {X 75.444,Y 66.007,Z 74.500,A 180.000,B 0.000,C 180.000} C_DIS
LIN {X 75.473,Y 65.969,Z 74.500,A 180.000,B 0.000,C 180.000} C_DIS
LIN {X 75.537,Y 65.880,Z 74.500,A 180.000,B 0.000,C 180.000} C_DIS
LIN {X 75.595,Y 65.791,Z 74.500,A 180.000,B 0.000,C 180.000} C_DIS
LIN {X 75.623,Y 65.744,Z 74.500,A 180.000,B 0.000,C 180.000} C_DIS
LIN {X 75.696,Y 65.612,Z 74.500,A 180.000,B 0.000,C 180.000} C_DIS
LIN {X 75.778,Y 65.433,Z 74.500,A 180.000,B 0.000,C 180.000} C_DIS
LIN {X 75.802,Y 65.375,Z 74.500,A 180.000,B 0.000,C 180.000} C_DIS
LIN {X 75.845,Y 65.254,Z 74.500,A 180.000,B 0.000,C 180.000} C_DIS
LIN {X 75.896,Y 65.075,Z 74.500,A 180.000,B 0.000,C 180.000} C_DIS
LIN {X 75.934,Y 64.897,Z 74.500,A 180.000,B 0.000,C 180.000} C_DIS
LIN {X 75.958,Y 64.718,Z 74.500,A 180.000,B 0.000,C 180.000} C_DIS
LIN {X 75.969,Y 64.539,Z 74.500,A 180.000,B 0.000,C 180.000} C_DIS
LIN {X 75.967,Y 64.360,Z 74.500,A 180.000,B 0.000,C 180.000} C_DIS
LIN {X 75.953,Y 64.182,Z 74.500,A 180.000,B 0.000,C 180.000} C_DIS
LIN {X 75.925,Y 64.003,Z 74.500,A 180.000,B 0.000,C 180.000} C_DIS
LIN {X 75.884,Y 63.824,Z 74.500,A 180.000,B 0.000,C 180.000} C_DIS
LIN {X 75.829,Y 63.645,Z 74.500,A 180.000,B 0.000,C 180.000} C_DIS
LIN {X 73.566,Y 56.936,Z 74.500,A 180.000,B 0.000,C 180.000} C_DIS
; Link Move Starts
LIN {X 73.471,Y 56.636,Z 74.500,A 180.000,B 0.000,C 180.000} C_DIS
LIN {X 73.371,Y 56.337,Z 74.499,A 180.000,B 0.000,C 180.000} C_DIS
LIN {X 73.272,Y 56.038,Z 74.498,A 180.000,B 0.000,C 180.000} C_DIS
LIN {X 73.173,Y 55.739,Z 74.496,A 180.000,B 0.000,C 180.000} C_DIS
LIN {X 73.075,Y 55.440,Z 74.494,A 180.000,B 0.000,C 180.000} C_DIS
LIN {X 72.977,Y 55.140,Z 74.491,A 180.000,B 0.000,C 180.000} C_DIS
LIN {X 72.880,Y 54.841,Z 74.488,A 180.000,B 0.000,C 180.000} C_DIS
LIN {X 72.783,Y 54.541,Z 74.485,A 180.000,B 0.000,C 180.000} C_DIS
LIN {X 72.687,Y 54.241,Z 74.481,A 180.000,B 0.000,C 180.000} C_DIS
LIN {X 72.591,Y 53.941,Z 74.477,A 180.000,B 0.000,C 180.000} C_DIS
LIN {X 72.496,Y 53.640,Z 74.472,A 180.000,B 0.000,C 180.000} C_DIS
LIN {X 72.448,Y 53.490,Z 74.469,A 180.000,B 0.000,C 180.000} C_DIS
LIN {X 72.401,Y 53.340,Z 74.467,A 180.000,B 0.000,C 180.000} C_DIS
LIN {X 72.353,Y 53.190,Z 74.464,A 180.000,B 0.000,C 180.000} C_DIS
LIN {X 72.306,Y 53.039,Z 74.461,A 180.000,B 0.000,C 180.000} C_DIS
LIN {X 72.259,Y 52.889,Z 74.459,A 180.000,B 0.000,C 180.000} C_DIS
LIN {X 72.212,Y 52.739,Z 74.456,A 180.000,B 0.000,C 180.000} C_DIS
LIN {X 72.165,Y 52.588,Z 74.452,A 180.000,B 0.000,C 180.000} C_DIS
LIN {X 72.119,Y 52.438,Z 74.449,A 180.000,B 0.000,C 180.000} C_DIS
LIN {X 72.072,Y 52.287,Z 74.446,A 180.000,B 0.000,C 180.000} C_DIS
LIN {X 72.025,Y 52.137,Z 74.443,A 180.000,B 0.000,C 180.000} C_DIS
LIN {X 71.979,Y 51.986,Z 74.439,A 180.000,B 0.000,C 180.000} C_DIS
LIN {X 71.933,Y 51.836,Z 74.436,A 180.000,B 0.000,C 180.000} C_DIS
LIN {X 71.886,Y 51.685,Z 74.432,A 180.000,B 0.000,C 180.000} C_DIS
LIN {X 71.840,Y 51.534,Z 74.428,A 180.000,B 0.000,C 180.000} C_DIS
LIN {X 71.794,Y 51.384,Z 74.425,A 180.000,B 0.000,C 180.000} C_DIS
LIN {X 71.748,Y 51.233,Z 74.421,A 180.000,B 0.000,C 180.000} C_DIS
LIN {X 71.702,Y 51.082,Z 74.417,A 180.000,B 0.000,C 180.000} C_DIS
LIN {X 71.657,Y 50.931,Z 74.413,A 180.000,B 0.000,C 180.000} C_DIS
LIN {X 71.611,Y 50.781,Z 74.409,A 180.000,B 0.000,C 180.000} C_DIS
LIN {X 71.565,Y 50.630,Z 74.405,A 180.000,B 0.000,C 180.000} C_DIS
LIN {X 71.520,Y 50.479,Z 74.400,A 180.000,B 0.000,C 180.000} C_DIS
LIN {X 71.474,Y 50.328,Z 74.396,A 180.000,B 0.000,C 180.000} C_DIS
LIN {X 71.429,Y 50.177,Z 74.392,A 180.000,B 0.000,C 180.000} C_DIS
LIN {X 71.384,Y 50.026,Z 74.387,A 180.000,B 0.000,C 180.000} C_DIS
LIN {X 71.339,Y 49.875,Z 74.383,A 180.000,B 0.000,C 180.000} C_DIS
LIN {X 71.294,Y 49.724,Z 74.378,A 180.000,B 0.000,C 180.000} C_DIS
LIN {X 71.249,Y 49.573,Z 74.373,A 180.000,B 0.000,C 180.000} C_DIS
LIN {X 71.204,Y 49.422,Z 74.369,A 180.000,B 0.000,C 180.000} C_DIS
LIN {X 71.159,Y 49.271,Z 74.364,A 180.000,B 0.000,C 180.000} C_DIS
LIN {X 71.114,Y 49.120,Z 74.359,A 180.000,B 0.000,C 180.000} C_DIS
LIN {X 71.069,Y 48.969,Z 74.354,A 180.000,B 0.000,C 180.000} C_DIS
LIN {X 71.047,Y 48.893,Z 74.351,A 180.000,B 0.000,C 180.000} C_DIS
LIN {X 71.025,Y 48.818,Z 74.349,A 180.000,B 0.000,C 180.000} C_DIS
LIN {X 71.002,Y 48.742,Z 74.346,A 180.000,B 0.000,C 180.000} C_DIS
LIN {X 70.980,Y 48.666,Z 74.344,A 180.000,B 0.000,C 180.000} C_DIS
LIN {X 70.958,Y 48.591,Z 74.341,A 180.000,B 0.000,C 180.000} C_DIS
LIN {X 70.936,Y 48.515,Z 74.339,A 180.000,B 0.000,C 180.000} C_DIS
LIN {X 70.913,Y 48.440,Z 74.336,A 180.000,B 0.000,C 180.000} C_DIS
LIN {X 70.891,Y 48.364,Z 74.333,A 180.000,B 0.000,C 180.000} C_DIS
LIN {X 70.869,Y 48.288,Z 74.331,A 180.000,B 0.000,C 180.000} C_DIS
LIN {X 70.847,Y 48.213,Z 74.328,A 180.000,B 0.000,C 180.000} C_DIS
LIN {X 70.825,Y 48.137,Z 74.325,A 180.000,B 0.000,C 180.000} C_DIS
LIN {X 70.803,Y 48.061,Z 74.323,A 180.000,B 0.000,C 180.000} C_DIS
LIN {X 70.780,Y 47.986,Z 74.320,A 180.000,B 0.000,C 180.000} C_DIS
LIN {X 70.758,Y 47.910,Z 74.317,A 180.000,B 0.000,C 180.000} C_DIS
LIN {X 70.736,Y 47.834,Z 74.315,A 180.000,B 0.000,C 180.000} C_DIS
LIN {X 70.714,Y 47.759,Z 74.312,A 180.000,B 0.000,C 180.000} C_DIS
LIN {X 70.692,Y 47.683,Z 74.309,A 180.000,B 0.000,C 180.000} C_DIS
LIN {X 70.670,Y 47.607,Z 74.307,A 180.000,B 0.000,C 180.000} C_DIS
LIN {X 70.648,Y 47.532,Z 74.304,A 180.000,B 0.000,C 180.000} C_DIS
LIN {X 70.626,Y 47.456,Z 74.301,A 180.000,B 0.000,C 180.000} C_DIS
LIN {X 70.604,Y 47.380,Z 74.298,A 180.000,B 0.000,C 180.000} C_DIS
LIN {X 70.582,Y 47.305,Z 74.295,A 180.000,B 0.000,C 180.000} C_DIS
LIN {X 70.560,Y 47.229,Z 74.293,A 180.000,B 0.000,C 180.000} C_DIS
LIN {X 70.538,Y 47.153,Z 74.290,A 180.000,B 0.000,C 180.000} C_DIS
LIN {X 70.516,Y 47.078,Z 74.287,A 180.000,B 0.000,C 180.000} C_DIS
LIN {X 70.494,Y 47.002,Z 74.284,A 180.000,B 0.000,C 180.000} C_DIS
LIN {X 70.472,Y 46.926,Z 74.282,A 180.000,B 0.000,C 180.000} C_DIS
LIN {X 70.450,Y 46.851,Z 74.279,A 180.000,B 0.000,C 180.000} C_DIS
LIN {X 70.428,Y 46.775,Z 74.276,A 180.000,B 0.000,C 180.000} C_DIS
LIN {X 70.406,Y 46.699,Z 74.273,A 180.000,B 0.000,C 180.000} C_DIS
LIN {X 70.384,Y 46.624,Z 74.271,A 180.000,B 0.000,C 180.000} C_DIS
LIN {X 70.362,Y 46.548,Z 74.268,A 180.000,B 0.000,C 180.000} C_DIS
LIN {X 70.339,Y 46.472,Z 74.265,A 180.000,B 0.000,C 180.000} C_DIS
LIN {X 70.317,Y 46.397,Z 74.262,A 180.000,B 0.000,C 180.000} C_DIS
LIN {X 70.295,Y 46.321,Z 74.260,A 180.000,B 0.000,C 180.000} C_DIS
LIN {X 70.251,Y 46.170,Z 74.254,A 180.000,B 0.000,C 180.000} C_DIS
LIN {X 70.229,Y 46.094,Z 74.251,A 180.000,B 0.000,C 180.000} C_DIS
LIN {X 70.185,Y 45.943,Z 74.246,A 180.000,B 0.000,C 180.000} C_DIS
LIN {X 70.119,Y 45.716,Z 74.238,A 180.000,B 0.000,C 180.000} C_DIS
LIN {X 70.075,Y 45.564,Z 74.232,A 180.000,B 0.000,C 180.000} C_DIS
LIN {X 70.053,Y 45.489,Z 74.229,A 180.000,B 0.000,C 180.000} C_DIS
LIN {X 70.009,Y 45.337,Z 74.224,A 180.000,B 0.000,C 180.000} C_DIS
LIN {X 69.943,Y 45.110,Z 74.216,A 180.000,B 0.000,C 180.000} C_DIS
LIN {X 69.899,Y 44.959,Z 74.210,A 180.000,B 0.000,C 180.000} C_DIS
LIN {X 69.877,Y 44.883,Z 74.207,A 180.000,B 0.000,C 180.000} C_DIS
LIN {X 69.834,Y 44.735,Z 74.202,A 180.000,B 0.000,C 180.000} C_DIS
LIN {X 69.812,Y 44.661,Z 74.199,A 180.000,B 0.000,C 180.000} C_DIS
LIN {X 69.790,Y 44.587,Z 74.197,A 180.000,B 0.000,C 180.000} C_DIS
LIN {X 69.756,Y 44.482,Z 74.193,A 180.000,B 0.000,C 180.000} C_DIS
LIN {X 69.718,Y 44.378,Z 74.189,A 180.000,B 0.000,C 180.000} C_DIS
LIN {X 69.683,Y 44.296,Z 74.186,A 180.000,B 0.000,C 180.000} C_DIS
LIN {X 69.645,Y 44.214,Z 74.183,A 180.000,B 0.000,C 180.000} C_DIS
LIN {X 69.590,Y 44.107,Z 74.178,A 180.000,B 0.000,C 180.000} C_DIS
LIN {X 69.529,Y 44.002,Z 74.174,A 180.000,B 0.000,C 180.000} C_DIS
LIN {X 69.474,Y 43.916,Z 74.171,A 180.000,B 0.000,C 180.000} C_DIS
LIN {X 69.415,Y 43.832,Z 74.167,A 180.000,B 0.000,C 180.000} C_DIS
LIN {X 69.352,Y 43.749,Z 74.163,A 180.000,B 0.000,C 180.000} C_DIS
LIN {X 69.285,Y 43.669,Z 74.160,A 180.000,B 0.000,C 180.000} C_DIS
LIN {X 69.200,Y 43.578,Z 74.155,A 180.000,B 0.000,C 180.000} C_DIS
LIN {X 69.111,Y 43.490,Z 74.151,A 180.000,B 0.000,C 180.000} C_DIS
LIN {X 69.022,Y 43.412,Z 74.147,A 180.000,B 0.000,C 180.000} C_DIS
LIN {X 68.930,Y 43.338,Z 74.143,A 180.000,B 0.000,C 180.000} C_DIS
LIN {X 68.823,Y 43.262,Z 74.138,A 180.000,B 0.000,C 180.000} C_DIS
LIN {X 68.712,Y 43.192,Z 74.134,A 180.000,B 0.000,C 180.000} C_DIS
LIN {X 68.594,Y 43.126,Z 74.129,A 180.000,B 0.000,C 180.000} C_DIS
LIN {X 68.472,Y 43.067,Z 74.124,A 180.000,B 0.000,C 180.000} C_DIS
LIN {X 68.343,Y 43.014,Z 74.119,A 180.000,B 0.000,C 180.000} C_DIS
LIN {X 68.211,Y 42.968,Z 74.114,A 180.000,B 0.000,C 180.000} C_DIS
LIN {X 68.141,Y 42.947,Z 74.112,A 180.000,B 0.000,C 180.000} C_DIS
LIN {X 68.069,Y 42.928,Z 74.109,A 180.000,B 0.000,C 180.000} C_DIS
LIN {X 67.998,Y 42.912,Z 74.107,A 180.000,B 0.000,C 180.000} C_DIS
LIN {X 67.925,Y 42.898,Z 74.104,A 180.000,B 0.000,C 180.000} C_DIS
LIN {X 67.850,Y 42.886,Z 74.102,A 180.000,B 0.000,C 180.000} C_DIS
LIN {X 67.774,Y 42.876,Z 74.099,A 180.000,B 0.000,C 180.000} C_DIS
LIN {X 67.697,Y 42.869,Z 74.096,A 180.000,B 0.000,C 180.000} C_DIS
LIN {X 67.621,Y 42.864,Z 74.093,A 180.000,B 0.000,C 180.000} C_DIS
LIN {X 67.541,Y 42.862,Z 74.091,A 180.000,B 0.000,C 180.000} C_DIS
LIN {X 67.460,Y 42.863,Z 74.088,A 180.000,B 0.000,C 180.000} C_DIS
LIN {X 67.380,Y 42.866,Z 74.085,A 180.000,B 0.000,C 180.000} C_DIS
LIN {X 67.300,Y 42.873,Z 74.082,A 180.000,B 0.000,C 180.000} C_DIS
LIN {X 67.221,Y 42.882,Z 74.080,A 180.000,B 0.000,C 180.000} C_DIS
LIN {X 67.142,Y 42.893,Z 74.077,A 180.000,B 0.000,C 180.000} C_DIS
LIN {X 67.064,Y 42.908,Z 74.074,A 180.000,B 0.000,C 180.000} C_DIS
LIN {X 66.986,Y 42.925,Z 74.071,A 180.000,B 0.000,C 180.000} C_DIS
LIN {X 66.909,Y 42.945,Z 74.068,A 180.000,B 0.000,C 180.000} C_DIS
LIN {X 66.834,Y 42.967,Z 74.066,A 180.000,B 0.000,C 180.000} C_DIS
LIN {X 66.759,Y 42.992,Z 74.063,A 180.000,B 0.000,C 180.000} C_DIS
LIN {X 66.087,Y 43.218,Z 74.038,A 180.000,B 0.000,C 180.000} C_DIS
LIN {X 65.266,Y 43.495,Z 74.008,A 180.000,B 0.000,C 180.000} C_DIS
LIN {X 62.879,Y 44.301,Z 73.920,A 180.000,B 0.000,C 180.000} C_DIS
LIN {X 62.506,Y 44.426,Z 73.906,A 180.000,B 0.000,C 180.000} C_DIS
LIN {X 62.282,Y 44.502,Z 73.898,A 180.000,B 0.000,C 180.000} C_DIS
LIN {X 62.058,Y 44.578,Z 73.890,A 180.000,B 0.000,C 180.000} C_DIS
LIN {X 61.312,Y 44.829,Z 73.862,A 180.000,B 0.000,C 180.000} C_DIS
LIN {X 61.088,Y 44.905,Z 73.854,A 180.000,B 0.000,C 180.000} C_DIS
LIN {X 60.939,Y 44.955,Z 73.848,A 180.000,B 0.000,C 180.000} C_DIS
LIN {X 60.491,Y 45.106,Z 73.832,A 180.000,B 0.000,C 180.000} C_DIS
LIN {X 60.416,Y 45.131,Z 73.829,A 180.000,B 0.000,C 180.000} C_DIS
LIN {X 60.267,Y 45.182,Z 73.824,A 180.000,B 0.000,C 180.000} C_DIS
LIN {X 59.819,Y 45.333,Z 73.807,A 180.000,B 0.000,C 180.000} C_DIS
LIN {X 59.670,Y 45.383,Z 73.802,A 180.000,B 0.000,C 180.000} C_DIS
LIN {X 59.222,Y 45.534,Z 73.785,A 180.000,B 0.000,C 180.000} C_DIS
LIN {X 59.073,Y 45.584,Z 73.780,A 180.000,B 0.000,C 180.000} C_DIS
LIN {X 58.849,Y 45.660,Z 73.771,A 180.000,B 0.000,C 180.000} C_DIS
LIN {X 58.700,Y 45.710,Z 73.766,A 180.000,B 0.000,C 180.000} C_DIS
LIN {X 58.625,Y 45.735,Z 73.763,A 180.000,B 0.000,C 180.000} C_DIS
LIN {X 58.476,Y 45.786,Z 73.758,A 180.000,B 0.000,C 180.000} C_DIS
LIN {X 58.252,Y 45.861,Z 73.749,A 180.000,B 0.000,C 180.000} C_DIS
LIN {X 58.103,Y 45.912,Z 73.744,A 180.000,B 0.000,C 180.000} C_DIS
LIN {X 58.028,Y 45.937,Z 73.741,A 180.000,B 0.000,C 180.000} C_DIS
LIN {X 57.879,Y 45.987,Z 73.736,A 180.000,B 0.000,C 180.000} C_DIS
LIN {X 57.655,Y 46.063,Z 73.727,A 180.000,B 0.000,C 180.000} C_DIS
LIN {X 57.506,Y 46.113,Z 73.722,A 180.000,B 0.000,C 180.000} C_DIS
LIN {X 57.432,Y 46.138,Z 73.719,A 180.000,B 0.000,C 180.000} C_DIS
LIN {X 57.282,Y 46.189,Z 73.714,A 180.000,B 0.000,C 180.000} C_DIS
LIN {X 57.058,Y 46.264,Z 73.705,A 180.000,B 0.000,C 180.000} C_DIS
LIN {X 56.909,Y 46.314,Z 73.700,A 180.000,B 0.000,C 180.000} C_DIS
LIN {X 56.835,Y 46.340,Z 73.697,A 180.000,B 0.000,C 180.000} C_DIS
LIN {X 56.685,Y 46.390,Z 73.692,A 180.000,B 0.000,C 180.000} C_DIS
LIN {X 56.536,Y 46.440,Z 73.686,A 180.000,B 0.000,C 180.000} C_DIS
LIN {X 56.387,Y 46.491,Z 73.681,A 180.000,B 0.000,C 180.000} C_DIS
LIN {X 56.238,Y 46.541,Z 73.675,A 180.000,B 0.000,C 180.000} C_DIS
LIN {X 56.088,Y 46.591,Z 73.670,A 180.000,B 0.000,C 180.000} C_DIS
LIN {X 55.939,Y 46.642,Z 73.665,A 180.000,B 0.000,C 180.000} C_DIS
LIN {X 55.865,Y 46.667,Z 73.662,A 180.000,B 0.000,C 180.000} C_DIS
LIN {X 55.790,Y 46.692,Z 73.660,A 180.000,B 0.000,C 180.000} C_DIS
LIN {X 55.715,Y 46.717,Z 73.657,A 180.000,B 0.000,C 180.000} C_DIS
LIN {X 55.641,Y 46.742,Z 73.655,A 180.000,B 0.000,C 180.000} C_DIS
LIN {X 55.566,Y 46.768,Z 73.652,A 180.000,B 0.000,C 180.000} C_DIS
LIN {X 55.491,Y 46.793,Z 73.649,A 180.000,B 0.000,C 180.000} C_DIS
LIN {X 55.342,Y 46.843,Z 73.644,A 180.000,B 0.000,C 180.000} C_DIS
LIN {X 55.193,Y 46.893,Z 73.640,A 180.000,B 0.000,C 180.000} C_DIS
LIN {X 55.044,Y 46.944,Z 73.635,A 180.000,B 0.000,C 180.000} C_DIS
LIN {X 54.894,Y 46.994,Z 73.630,A 180.000,B 0.000,C 180.000} C_DIS
LIN {X 54.745,Y 47.044,Z 73.625,A 180.000,B 0.000,C 180.000} C_DIS
LIN {X 54.596,Y 47.095,Z 73.620,A 180.000,B 0.000,C 180.000} C_DIS
LIN {X 54.447,Y 47.145,Z 73.616,A 180.000,B 0.000,C 180.000} C_DIS
LIN {X 54.298,Y 47.195,Z 73.611,A 180.000,B 0.000,C 180.000} C_DIS
LIN {X 54.148,Y 47.246,Z 73.607,A 180.000,B 0.000,C 180.000} C_DIS
LIN {X 53.999,Y 47.296,Z 73.603,A 180.000,B 0.000,C 180.000} C_DIS
LIN {X 53.850,Y 47.346,Z 73.598,A 180.000,B 0.000,C 180.000} C_DIS
LIN {X 53.701,Y 47.397,Z 73.594,A 180.000,B 0.000,C 180.000} C_DIS
LIN {X 53.551,Y 47.447,Z 73.590,A 180.000,B 0.000,C 180.000} C_DIS
LIN {X 53.402,Y 47.498,Z 73.586,A 180.000,B 0.000,C 180.000} C_DIS
LIN {X 53.253,Y 47.548,Z 73.582,A 180.000,B 0.000,C 180.000} C_DIS
LIN {X 53.104,Y 47.598,Z 73.578,A 180.000,B 0.000,C 180.000} C_DIS
LIN {X 52.954,Y 47.649,Z 73.574,A 180.000,B 0.000,C 180.000} C_DIS
LIN {X 52.805,Y 47.699,Z 73.570,A 180.000,B 0.000,C 180.000} C_DIS
LIN {X 52.656,Y 47.749,Z 73.567,A 180.000,B 0.000,C 180.000} C_DIS
LIN {X 52.507,Y 47.800,Z 73.563,A 180.000,B 0.000,C 180.000} C_DIS
LIN {X 52.357,Y 47.850,Z 73.560,A 180.000,B 0.000,C 180.000} C_DIS
LIN {X 52.208,Y 47.900,Z 73.556,A 180.000,B 0.000,C 180.000} C_DIS
LIN {X 52.059,Y 47.951,Z 73.553,A 180.000,B 0.000,C 180.000} C_DIS
LIN {X 51.910,Y 48.001,Z 73.550,A 180.000,B 0.000,C 180.000} C_DIS
LIN {X 51.761,Y 48.051,Z 73.547,A 180.000,B 0.000,C 180.000} C_DIS
LIN {X 51.611,Y 48.102,Z 73.543,A 180.000,B 0.000,C 180.000} C_DIS
LIN {X 51.462,Y 48.152,Z 73.541,A 180.000,B 0.000,C 180.000} C_DIS
LIN {X 51.313,Y 48.202,Z 73.538,A 180.000,B 0.000,C 180.000} C_DIS
LIN {X 51.164,Y 48.253,Z 73.535,A 180.000,B 0.000,C 180.000} C_DIS
LIN {X 51.014,Y 48.303,Z 73.532,A 180.000,B 0.000,C 180.000} C_DIS
LIN {X 50.865,Y 48.353,Z 73.530,A 180.000,B 0.000,C 180.000} C_DIS
LIN {X 50.567,Y 48.454,Z 73.525,A 180.000,B 0.000,C 180.000} C_DIS
LIN {X 50.268,Y 48.555,Z 73.520,A 180.000,B 0.000,C 180.000} C_DIS
LIN {X 49.970,Y 48.655,Z 73.516,A 180.000,B 0.000,C 180.000} C_DIS
LIN {X 49.671,Y 48.756,Z 73.513,A 180.000,B 0.000,C 180.000} C_DIS
LIN {X 49.373,Y 48.857,Z 73.510,A 180.000,B 0.000,C 180.000} C_DIS
LIN {X 49.074,Y 48.958,Z 73.507,A 180.000,B 0.000,C 180.000} C_DIS
LIN {X 48.776,Y 49.058,Z 73.505,A 180.000,B 0.000,C 180.000} C_DIS
LIN {X 48.477,Y 49.159,Z 73.503,A 180.000,B 0.000,C 180.000} C_DIS
LIN {X 48.179,Y 49.260,Z 73.501,A 180.000,B 0.000,C 180.000} C_DIS
LIN {X 47.880,Y 49.360,Z 73.500,A 180.000,B 0.000,C 180.000} C_DIS
LIN {X 47.582,Y 49.461,Z 73.500,A 180.000,B 0.000,C 180.000} C_DIS
LIN {X 47.482,Y 49.495,Z 73.500,A 180.000,B 0.000,C 180.000} C_DIS
; Cutting Move Starts
LIN {X 45.590,Y 50.133,Z 73.500,A 180.000,B 0.000,C 180.000} C_DIS
LIN {X 45.411,Y 50.194,Z 73.500,A 180.000,B 0.000,C 180.000} C_DIS
LIN {X 45.296,Y 50.238,Z 73.500,A 180.000,B 0.000,C 180.000} C_DIS
LIN {X 45.232,Y 50.265,Z 73.500,A 180.000,B 0.000,C 180.000} C_DIS
LIN {X 45.053,Y 50.353,Z 73.500,A 180.000,B 0.000,C 180.000} C_DIS
LIN {X 44.944,Y 50.416,Z 73.500,A 180.000,B 0.000,C 180.000} C_DIS
LIN {X 44.874,Y 50.461,Z 73.500,A 180.000,B 0.000,C 180.000} C_DIS
LIN {X 44.785,Y 50.522,Z 73.500,A 180.000,B 0.000,C 180.000} C_DIS
LIN {X 44.696,Y 50.590,Z 73.500,A 180.000,B 0.000,C 180.000} C_DIS
LIN {X 44.689,Y 50.595,Z 73.500,A 180.000,B 0.000,C 180.000} C_DIS
LIN {X 44.603,Y 50.667,Z 73.500,A 180.000,B 0.000,C 180.000} C_DIS
LIN {X 44.517,Y 50.746,Z 73.500,A 180.000,B 0.000,C 180.000} C_DIS
LIN {X 44.488,Y 50.774,Z 73.500,A 180.000,B 0.000,C 180.000} C_DIS
LIN {X 44.410,Y 50.855,Z 73.500,A 180.000,B 0.000,C 180.000} C_DIS
LIN {X 44.338,Y 50.936,Z 73.500,A 180.000,B 0.000,C 180.000} C_DIS
LIN {X 44.325,Y 50.953,Z 73.500,A 180.000,B 0.000,C 180.000} C_DIS
LIN {X 44.254,Y 51.042,Z 73.500,A 180.000,B 0.000,C 180.000} C_DIS
LIN {X 44.189,Y 51.131,Z 73.500,A 180.000,B 0.000,C 180.000} C_DIS
LIN {X 44.159,Y 51.176,Z 73.500,A 180.000,B 0.000,C 180.000} C_DIS
LIN {X 44.077,Y 51.310,Z 73.500,A 180.000,B 0.000,C 180.000} C_DIS
LIN {X 43.984,Y 51.489,Z 73.500,A 180.000,B 0.000,C 180.000} C_DIS
LIN {X 43.981,Y 51.497,Z 73.500,A 180.000,B 0.000,C 180.000} C_DIS
LIN {X 43.909,Y 51.668,Z 73.500,A 180.000,B 0.000,C 180.000} C_DIS
LIN {X 43.849,Y 51.847,Z 73.500,A 180.000,B 0.000,C 180.000} C_DIS
LIN {X 43.804,Y 52.025,Z 73.500,A 180.000,B 0.000,C 180.000} C_DIS
LIN {X 43.802,Y 52.035,Z 73.500,A 180.000,B 0.000,C 180.000} C_DIS
LIN {X 43.772,Y 52.204,Z 73.500,A 180.000,B 0.000,C 180.000} C_DIS
LIN {X 43.754,Y 52.383,Z 73.500,A 180.000,B 0.000,C 180.000} C_DIS
LIN {X 43.748,Y 52.562,Z 73.500,A 180.000,B 0.000,C 180.000} C_DIS
LIN {X 43.756,Y 52.740,Z 73.500,A 180.000,B 0.000,C 180.000} C_DIS
LIN {X 43.776,Y 52.919,Z 73.500,A 180.000,B 0.000,C 180.000} C_DIS
LIN {X 43.802,Y 53.064,Z 73.500,A 180.000,B 0.000,C 180.000} C_DIS
LIN {X 43.809,Y 53.098,Z 73.500,A 180.000,B 0.000,C 180.000} C_DIS
LIN {X 43.856,Y 53.277,Z 73.500,A 180.000,B 0.000,C 180.000} C_DIS
LIN {X 43.916,Y 53.455,Z 73.500,A 180.000,B 0.000,C 180.000} C_DIS
LIN {X 50.248,Y 72.226,Z 73.500,A 180.000,B 0.000,C 180.000} C_DIS
LIN {X 50.311,Y 72.405,Z 73.500,A 180.000,B 0.000,C 180.000} C_DIS
LIN {X 50.388,Y 72.584,Z 73.500,A 180.000,B 0.000,C 180.000} C_DIS
LIN {X 50.416,Y 72.640,Z 73.500,A 180.000,B 0.000,C 180.000} C_DIS
LIN {X 50.484,Y 72.763,Z 73.500,A 180.000,B 0.000,C 180.000} C_DIS
LIN {X 50.595,Y 72.936,Z 73.500,A 180.000,B 0.000,C 180.000} C_DIS
LIN {X 50.599,Y 72.941,Z 73.500,A 180.000,B 0.000,C 180.000} C_DIS
LIN {X 50.665,Y 73.031,Z 73.500,A 180.000,B 0.000,C 180.000} C_DIS
LIN {X 50.737,Y 73.120,Z 73.500,A 180.000,B 0.000,C 180.000} C_DIS
LIN {X 50.774,Y 73.162,Z 73.500,A 180.000,B 0.000,C 180.000} C_DIS
LIN {X 50.905,Y 73.299,Z 73.500,A 180.000,B 0.000,C 180.000} C_DIS
LIN {X 50.953,Y 73.343,Z 73.500,A 180.000,B 0.000,C 180.000} C_DIS
LIN {X 51.112,Y 73.478,Z 73.500,A 180.000,B 0.000,C 180.000} C_DIS
LIN {X 51.131,Y 73.493,Z 73.500,A 180.000,B 0.000,C 180.000} C_DIS
LIN {X 51.310,Y 73.616,Z 73.500,A 180.000,B 0.000,C 180.000} C_DIS
LIN {X 51.376,Y 73.656,Z 73.500,A 180.000,B 0.000,C 180.000} C_DIS
LIN {X 51.489,Y 73.719,Z 73.500,A 180.000,B 0.000,C 180.000} C_DIS
LIN {X 51.668,Y 73.803,Z 73.500,A 180.000,B 0.000,C 180.000} C_DIS
LIN {X 51.749,Y 73.835,Z 73.500,A 180.000,B 0.000,C 180.000} C_DIS
LIN {X 51.847,Y 73.870,Z 73.500,A 180.000,B 0.000,C 180.000} C_DIS
LIN {X 52.025,Y 73.923,Z 73.500,A 180.000,B 0.000,C 180.000} C_DIS
LIN {X 52.204,Y 73.961,Z 73.500,A 180.000,B 0.000,C 180.000} C_DIS
LIN {X 52.383,Y 73.987,Z 73.500,A 180.000,B 0.000,C 180.000} C_DIS
LIN {X 52.562,Y 73.999,Z 73.500,A 180.000,B 0.000,C 180.000} C_DIS
LIN {X 52.740,Y 73.998,Z 73.500,A 180.000,B 0.000,C 180.000} C_DIS
LIN {X 52.919,Y 73.985,Z 73.500,A 180.000,B 0.000,C 180.000} C_DIS
LIN {X 53.098,Y 73.958,Z 73.500,A 180.000,B 0.000,C 180.000} C_DIS
